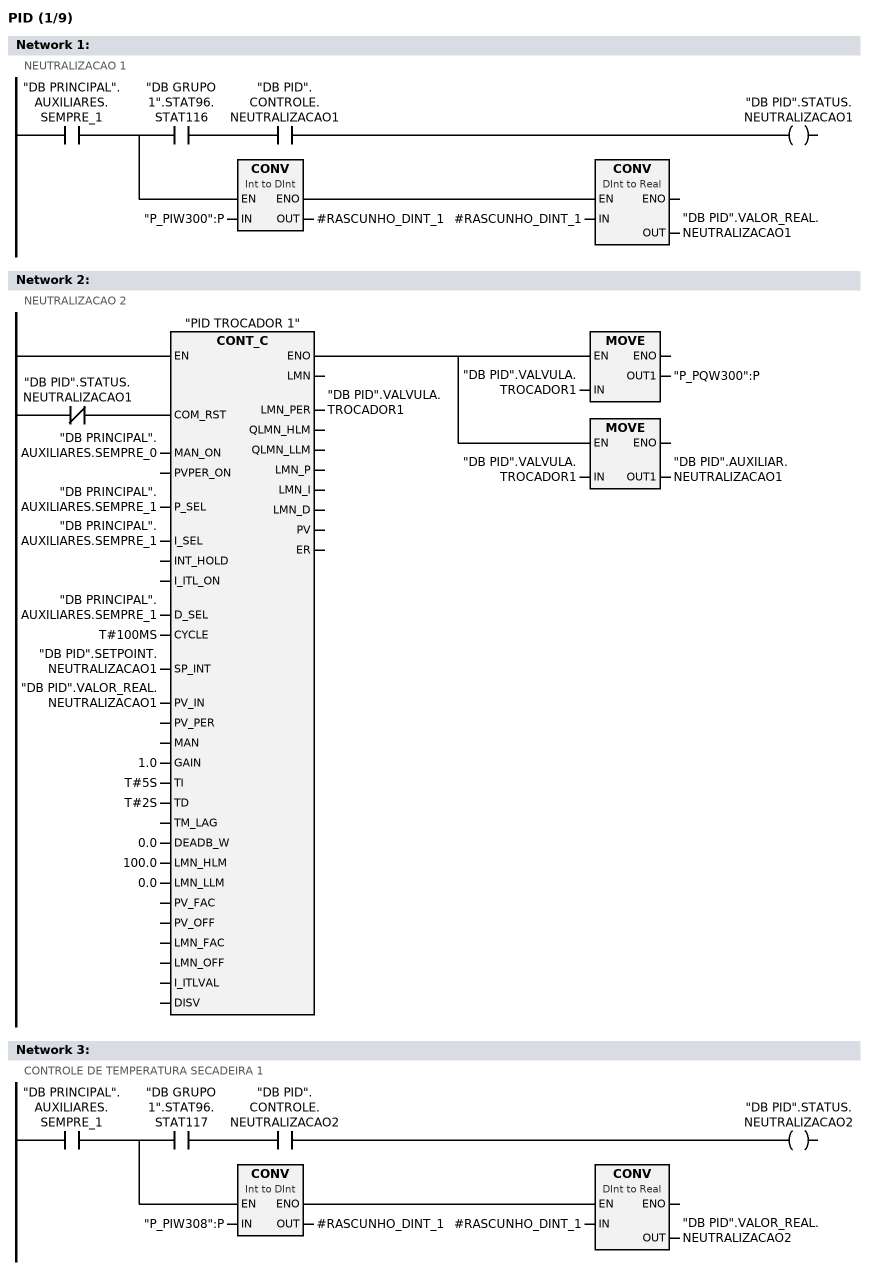
   RUNG wire#powerrail
      Contact( "DB PRINCIPAL".AUXILIARES.SEMPRE_1 )
      wire#w1
      Contact( "DB GRUPO 1".STAT96.STAT116 )
      Contact( "DB PID".CONTROLE.NEUTRALIZACAO1 )
      Coil( "DB PID".STATUS.NEUTRALIZACAO1 )
   END_RUNG
   RUNG wire#w1
      { S7_Templates := "[SrcType := Int, DestType := DInt]"; S7_GenerateENO := "TRUE" } Convert(in := "P_PIW300":P, out => #RASCUNHO_DINT_1)
      { S7_Templates := "[SrcType := DInt, DestType := Real]"; S7_GenerateENO := "TRUE" } Convert(in := #RASCUNHO_DINT_1, out => "DB PID".VALOR_REAL.NEUTRALIZACAO1)
   END_RUNG
   // the same network as SCL:
   // ENO of a box is taken as its EN; it also drops when the box reports an error
   "DB PID".STATUS.NEUTRALIZACAO1 := "DB PRINCIPAL".AUXILIARES.SEMPRE_1 AND "DB GRUPO 1".STAT96.STAT116 AND "DB PID".CONTROLE.NEUTRALIZACAO1;
   IF "DB PRINCIPAL".AUXILIARES.SEMPRE_1 THEN
       #RASCUNHO_DINT_1 := INT_TO_DINT("P_PIW300":P);
       "DB PID".VALOR_REAL.NEUTRALIZACAO1 := DINT_TO_REAL(#RASCUNHO_DINT_1);
   END_IF;
END_REGION

REGION Network 2
   // NEUTRALIZACAO 2
   // ENO of a box is taken as its EN; it also drops when the box reports an error
   "PID TROCADOR 1"(COM_RST := NOT "DB PID".STATUS.NEUTRALIZACAO1,   // CONT_C
                    MAN_ON := "DB PRINCIPAL".AUXILIARES.SEMPRE_0,
                    P_SEL := "DB PRINCIPAL".AUXILIARES.SEMPRE_1,
                    I_SEL := "DB PRINCIPAL".AUXILIARES.SEMPRE_1,
                    D_SEL := "DB PRINCIPAL".AUXILIARES.SEMPRE_1,
                    CYCLE := T#100MS,
                    SP_INT := "DB PID".SETPOINT.NEUTRALIZACAO1,
                    PV_IN := "DB PID".VALOR_REAL.NEUTRALIZACAO1,
                    GAIN := 1.0,
                    TI := T#5S,
                    TD := T#2S,
                    DEADB_W := 0.0,
                    LMN_HLM := 100.0,
                    LMN_LLM := 0.0,
                    LMN_PER => "DB PID".VALVULA.TROCADOR1);
   "P_PQW300":P := "DB PID".VALVULA.TROCADOR1;
   "DB PID".AUXILIAR.NEUTRALIZACAO1 := "DB PID".VALVULA.TROCADOR1;
END_REGION

REGION Network 3
   // CONTROLE DE TEMPERATURA SECADEIRA 1
   RUNG wire#powerrail
      Contact( "DB PRINCIPAL".AUXILIARES.SEMPRE_1 )
      wire#w1
      Contact( "DB GRUPO 1".STAT96.STAT117 )
      Contact( "DB PID".CONTROLE.NEUTRALIZACAO2 )
      Coil( "DB PID".STATUS.NEUTRALIZACAO2 )
   END_RUNG
   RUNG wire#w1
      { S7_Templates := "[SrcType := Int, DestType := DInt]"; S7_GenerateENO := "TRUE" } Convert(in := "P_PIW308":P, out => #RASCUNHO_DINT_1)
      { S7_Templates := "[SrcType := DInt, DestType := Real]"; S7_GenerateENO := "TRUE" } Convert(in := #RASCUNHO_DINT_1, out => "DB PID".VALOR_REAL.NEUTRALIZACAO2)
   END_RUNG
   // the same network as SCL:
   // ENO of a box is taken as its EN; it also drops when the box reports an error
   "DB PID".STATUS.NEUTRALIZACAO2 := "DB PRINCIPAL".AUXILIARES.SEMPRE_1 AND "DB GRUPO 1".STAT96.STAT117 AND "DB PID".CONTROLE.NEUTRALIZACAO2;
   IF "DB PRINCIPAL".AUXILIARES.SEMPRE_1 THEN
       #RASCUNHO_DINT_1 := INT_TO_DINT("P_PIW308":P);
       "DB PID".VALOR_REAL.NEUTRALIZACAO2 := DINT_TO_REAL(#RASCUNHO_DINT_1);
   END_IF;
END_REGION

REGION Network 4
   // CONTROLE DE TEMPERATURA SECADEIRA 2
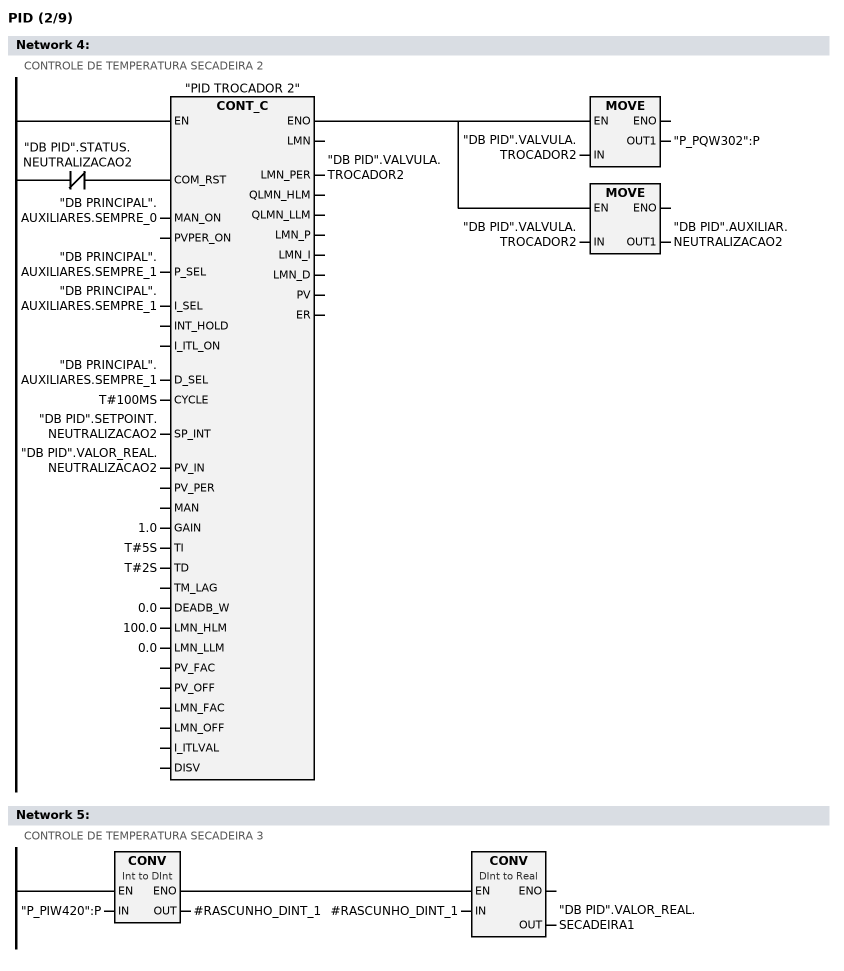
   // ENO of a box is taken as its EN; it also drops when the box reports an error
   "PID TROCADOR 2"(COM_RST := NOT "DB PID".STATUS.NEUTRALIZACAO2,   // CONT_C
                    MAN_ON := "DB PRINCIPAL".AUXILIARES.SEMPRE_0,
                    P_SEL := "DB PRINCIPAL".AUXILIARES.SEMPRE_1,
                    I_SEL := "DB PRINCIPAL".AUXILIARES.SEMPRE_1,
                    D_SEL := "DB PRINCIPAL".AUXILIARES.SEMPRE_1,
                    CYCLE := T#100MS,
                    SP_INT := "DB PID".SETPOINT.NEUTRALIZACAO2,
                    PV_IN := "DB PID".VALOR_REAL.NEUTRALIZACAO2,
                    GAIN := 1.0,
                    TI := T#5S,
                    TD := T#2S,
                    DEADB_W := 0.0,
                    LMN_HLM := 100.0,
                    LMN_LLM := 0.0,
                    LMN_PER => "DB PID".VALVULA.TROCADOR2);
   "P_PQW302":P := "DB PID".VALVULA.TROCADOR2;
   "DB PID".AUXILIAR.NEUTRALIZACAO2 := "DB PID".VALVULA.TROCADOR2;
END_REGION

REGION Network 5
   // CONTROLE DE TEMPERATURA SECADEIRA 3
   RUNG wire#powerrail
      { S7_Templates := "[SrcType := Int, DestType := DInt]"; S7_GenerateENO := "TRUE" } Convert(in := "P_PIW420":P, out => #RASCUNHO_DINT_1)
      { S7_Templates := "[SrcType := DInt, DestType := Real]"; S7_GenerateENO := "TRUE" } Convert(in := #RASCUNHO_DINT_1, out => "DB PID".VALOR_REAL.SECADEIRA1)
   END_RUNG
   // the same network as SCL:
   // ENO of a box is taken as its EN; it also drops when the box reports an error
   #RASCUNHO_DINT_1 := INT_TO_DINT("P_PIW420":P);
   "DB PID".VALOR_REAL.SECADEIRA1 := DINT_TO_REAL(#RASCUNHO_DINT_1);
END_REGION

REGION Network 6
   // CONTROLE DE TEMPERATURA SECADEIRA 4
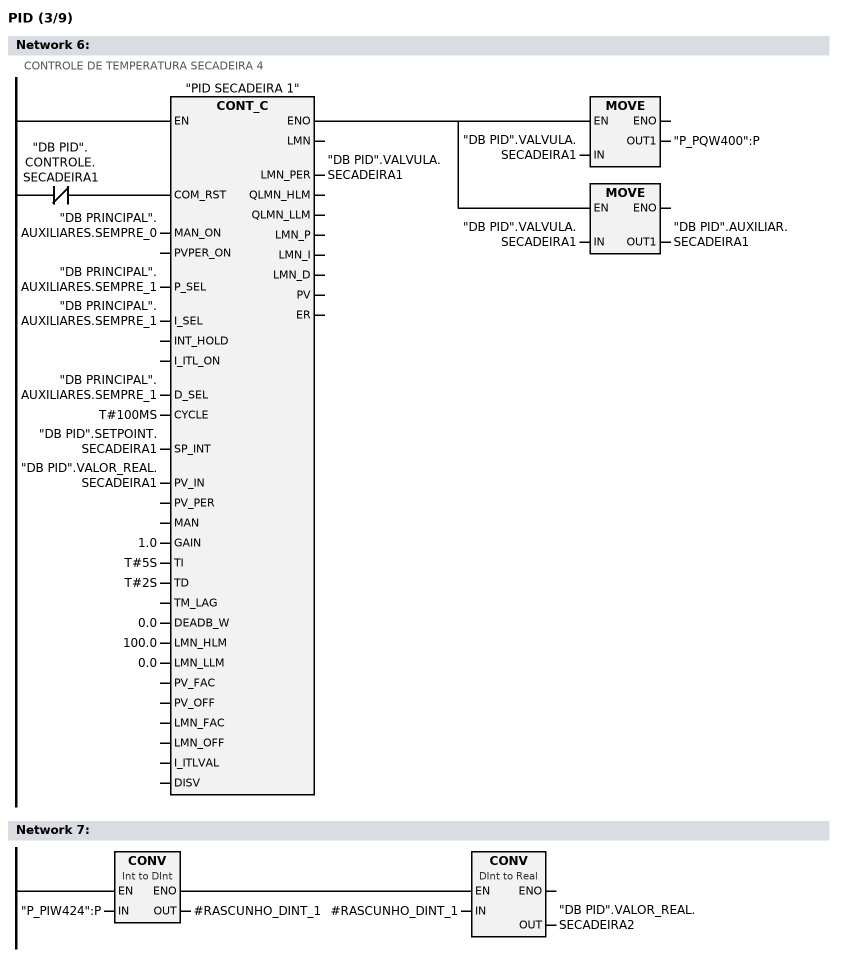
   // ENO of a box is taken as its EN; it also drops when the box reports an error
   "PID SECADEIRA 1"(COM_RST := NOT "DB PID".CONTROLE.SECADEIRA1,   // CONT_C
                     MAN_ON := "DB PRINCIPAL".AUXILIARES.SEMPRE_0,
                     P_SEL := "DB PRINCIPAL".AUXILIARES.SEMPRE_1,
                     I_SEL := "DB PRINCIPAL".AUXILIARES.SEMPRE_1,
                     D_SEL := "DB PRINCIPAL".AUXILIARES.SEMPRE_1,
                     CYCLE := T#100MS,
                     SP_INT := "DB PID".SETPOINT.SECADEIRA1,
                     PV_IN := "DB PID".VALOR_REAL.SECADEIRA1,
                     GAIN := 1.0,
                     TI := T#5S,
                     TD := T#2S,
                     DEADB_W := 0.0,
                     LMN_HLM := 100.0,
                     LMN_LLM := 0.0,
                     LMN_PER => "DB PID".VALVULA.SECADEIRA1);
   "P_PQW400":P := "DB PID".VALVULA.SECADEIRA1;
   "DB PID".AUXILIAR.SECADEIRA1 := "DB PID".VALVULA.SECADEIRA1;
END_REGION

REGION Network 7
   RUNG wire#powerrail
      { S7_Templates := "[SrcType := Int, DestType := DInt]"; S7_GenerateENO := "TRUE" } Convert(in := "P_PIW424":P, out => #RASCUNHO_DINT_1)
      { S7_Templates := "[SrcType := DInt, DestType := Real]"; S7_GenerateENO := "TRUE" } Convert(in := #RASCUNHO_DINT_1, out => "DB PID".VALOR_REAL.SECADEIRA2)
   END_RUNG
   // the same network as SCL:
   // ENO of a box is taken as its EN; it also drops when the box reports an error
   #RASCUNHO_DINT_1 := INT_TO_DINT("P_PIW424":P);
   "DB PID".VALOR_REAL.SECADEIRA2 := DINT_TO_REAL(#RASCUNHO_DINT_1);
END_REGION

REGION Network 8
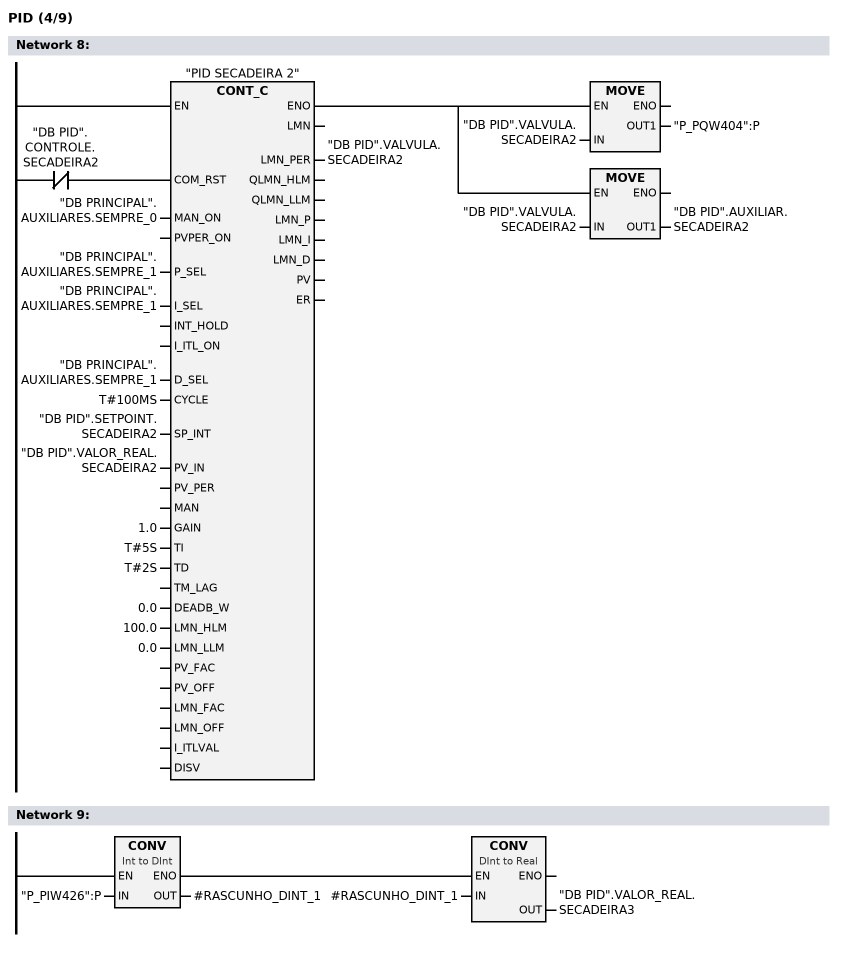
   // ENO of a box is taken as its EN; it also drops when the box reports an error
   "PID SECADEIRA 2"(COM_RST := NOT "DB PID".CONTROLE.SECADEIRA2,   // CONT_C
                     MAN_ON := "DB PRINCIPAL".AUXILIARES.SEMPRE_0,
                     P_SEL := "DB PRINCIPAL".AUXILIARES.SEMPRE_1,
                     I_SEL := "DB PRINCIPAL".AUXILIARES.SEMPRE_1,
                     D_SEL := "DB PRINCIPAL".AUXILIARES.SEMPRE_1,
                     CYCLE := T#100MS,
                     SP_INT := "DB PID".SETPOINT.SECADEIRA2,
                     PV_IN := "DB PID".VALOR_REAL.SECADEIRA2,
                     GAIN := 1.0,
                     TI := T#5S,
                     TD := T#2S,
                     DEADB_W := 0.0,
                     LMN_HLM := 100.0,
                     LMN_LLM := 0.0,
                     LMN_PER => "DB PID".VALVULA.SECADEIRA2);
   "P_PQW404":P := "DB PID".VALVULA.SECADEIRA2;
   "DB PID".AUXILIAR.SECADEIRA2 := "DB PID".VALVULA.SECADEIRA2;
END_REGION

REGION Network 9
   RUNG wire#powerrail
      { S7_Templates := "[SrcType := Int, DestType := DInt]"; S7_GenerateENO := "TRUE" } Convert(in := "P_PIW426":P, out => #RASCUNHO_DINT_1)
      { S7_Templates := "[SrcType := DInt, DestType := Real]"; S7_GenerateENO := "TRUE" } Convert(in := #RASCUNHO_DINT_1, out => "DB PID".VALOR_REAL.SECADEIRA3)
   END_RUNG
   // the same network as SCL:
   // ENO of a box is taken as its EN; it also drops when the box reports an error
   #RASCUNHO_DINT_1 := INT_TO_DINT("P_PIW426":P);
   "DB PID".VALOR_REAL.SECADEIRA3 := DINT_TO_REAL(#RASCUNHO_DINT_1);
END_REGION

REGION Network 10
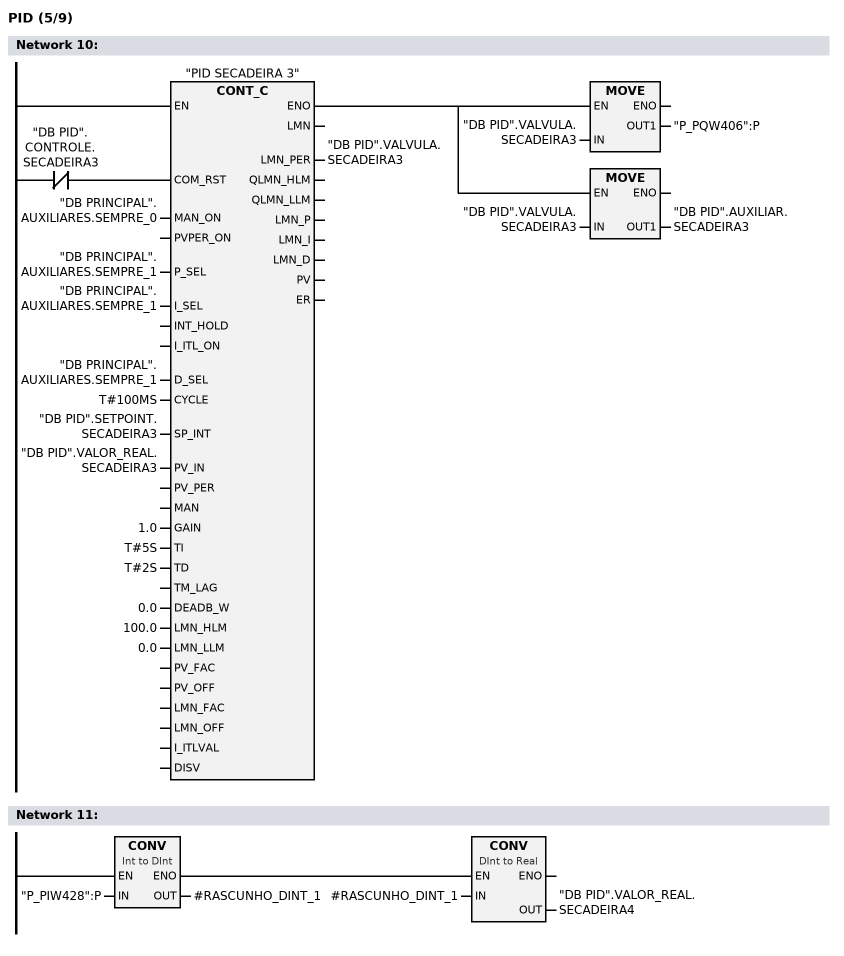
   // ENO of a box is taken as its EN; it also drops when the box reports an error
   "PID SECADEIRA 3"(COM_RST := NOT "DB PID".CONTROLE.SECADEIRA3,   // CONT_C
                     MAN_ON := "DB PRINCIPAL".AUXILIARES.SEMPRE_0,
                     P_SEL := "DB PRINCIPAL".AUXILIARES.SEMPRE_1,
                     I_SEL := "DB PRINCIPAL".AUXILIARES.SEMPRE_1,
                     D_SEL := "DB PRINCIPAL".AUXILIARES.SEMPRE_1,
                     CYCLE := T#100MS,
                     SP_INT := "DB PID".SETPOINT.SECADEIRA3,
                     PV_IN := "DB PID".VALOR_REAL.SECADEIRA3,
                     GAIN := 1.0,
                     TI := T#5S,
                     TD := T#2S,
                     DEADB_W := 0.0,
                     LMN_HLM := 100.0,
                     LMN_LLM := 0.0,
                     LMN_PER => "DB PID".VALVULA.SECADEIRA3);
   "P_PQW406":P := "DB PID".VALVULA.SECADEIRA3;
   "DB PID".AUXILIAR.SECADEIRA3 := "DB PID".VALVULA.SECADEIRA3;
END_REGION

REGION Network 11
   RUNG wire#powerrail
      { S7_Templates := "[SrcType := Int, DestType := DInt]"; S7_GenerateENO := "TRUE" } Convert(in := "P_PIW428":P, out => #RASCUNHO_DINT_1)
      { S7_Templates := "[SrcType := DInt, DestType := Real]"; S7_GenerateENO := "TRUE" } Convert(in := #RASCUNHO_DINT_1, out => "DB PID".VALOR_REAL.SECADEIRA4)
   END_RUNG
   // the same network as SCL:
   // ENO of a box is taken as its EN; it also drops when the box reports an error
   #RASCUNHO_DINT_1 := INT_TO_DINT("P_PIW428":P);
   "DB PID".VALOR_REAL.SECADEIRA4 := DINT_TO_REAL(#RASCUNHO_DINT_1);
END_REGION

REGION Network 12: PID SECADEIRA 4
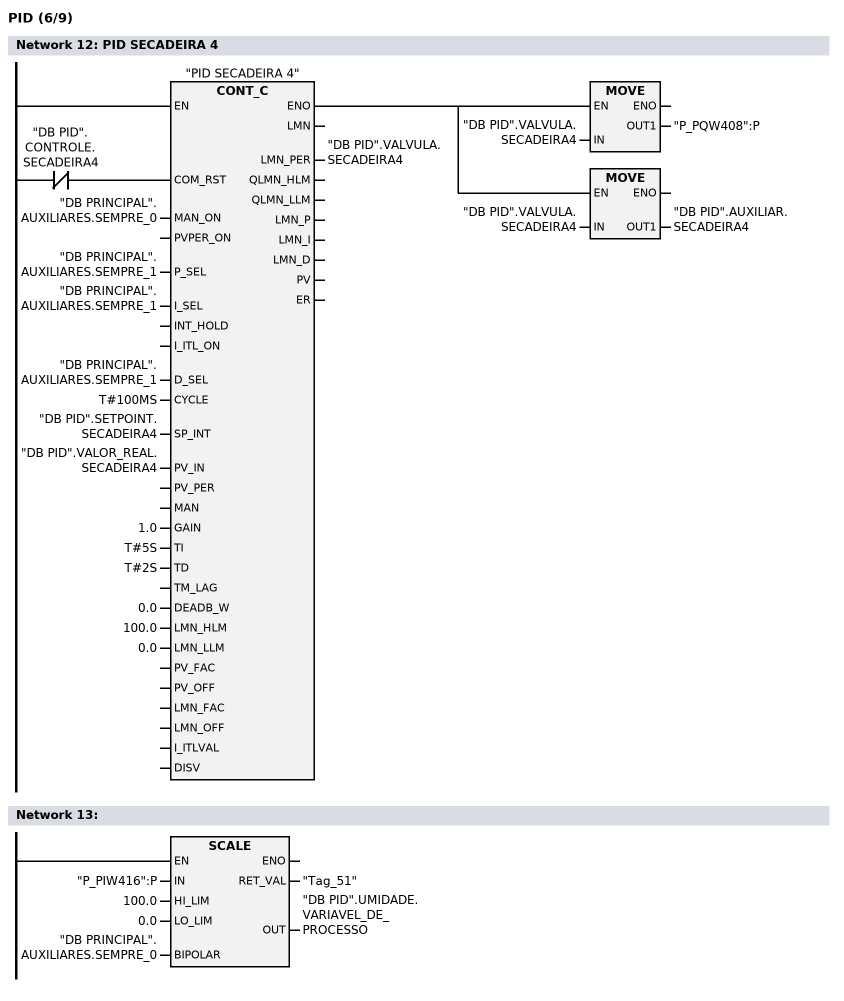
   // ENO of a box is taken as its EN; it also drops when the box reports an error
   "PID SECADEIRA 4"(COM_RST := NOT "DB PID".CONTROLE.SECADEIRA4,   // CONT_C
                     MAN_ON := "DB PRINCIPAL".AUXILIARES.SEMPRE_0,
                     P_SEL := "DB PRINCIPAL".AUXILIARES.SEMPRE_1,
                     I_SEL := "DB PRINCIPAL".AUXILIARES.SEMPRE_1,
                     D_SEL := "DB PRINCIPAL".AUXILIARES.SEMPRE_1,
                     CYCLE := T#100MS,
                     SP_INT := "DB PID".SETPOINT.SECADEIRA4,
                     PV_IN := "DB PID".VALOR_REAL.SECADEIRA4,
                     GAIN := 1.0,
                     TI := T#5S,
                     TD := T#2S,
                     DEADB_W := 0.0,
                     LMN_HLM := 100.0,
                     LMN_LLM := 0.0,
                     LMN_PER => "DB PID".VALVULA.SECADEIRA4);
   "P_PQW408":P := "DB PID".VALVULA.SECADEIRA4;
   "DB PID".AUXILIAR.SECADEIRA4 := "DB PID".VALVULA.SECADEIRA4;
END_REGION

REGION Network 13
   "Tag_51" := SCALE(IN := "P_PIW416":P,
                     HI_LIM := 100.0,
                     LO_LIM := 0.0,
                     BIPOLAR := "DB PRINCIPAL".AUXILIARES.SEMPRE_0,
                     OUT => "DB PID".UMIDADE.VARIAVEL_DE_PROCESSO);
END_REGION

REGION Network 14: PID SECADEIRA 4 - Controle de Umidade
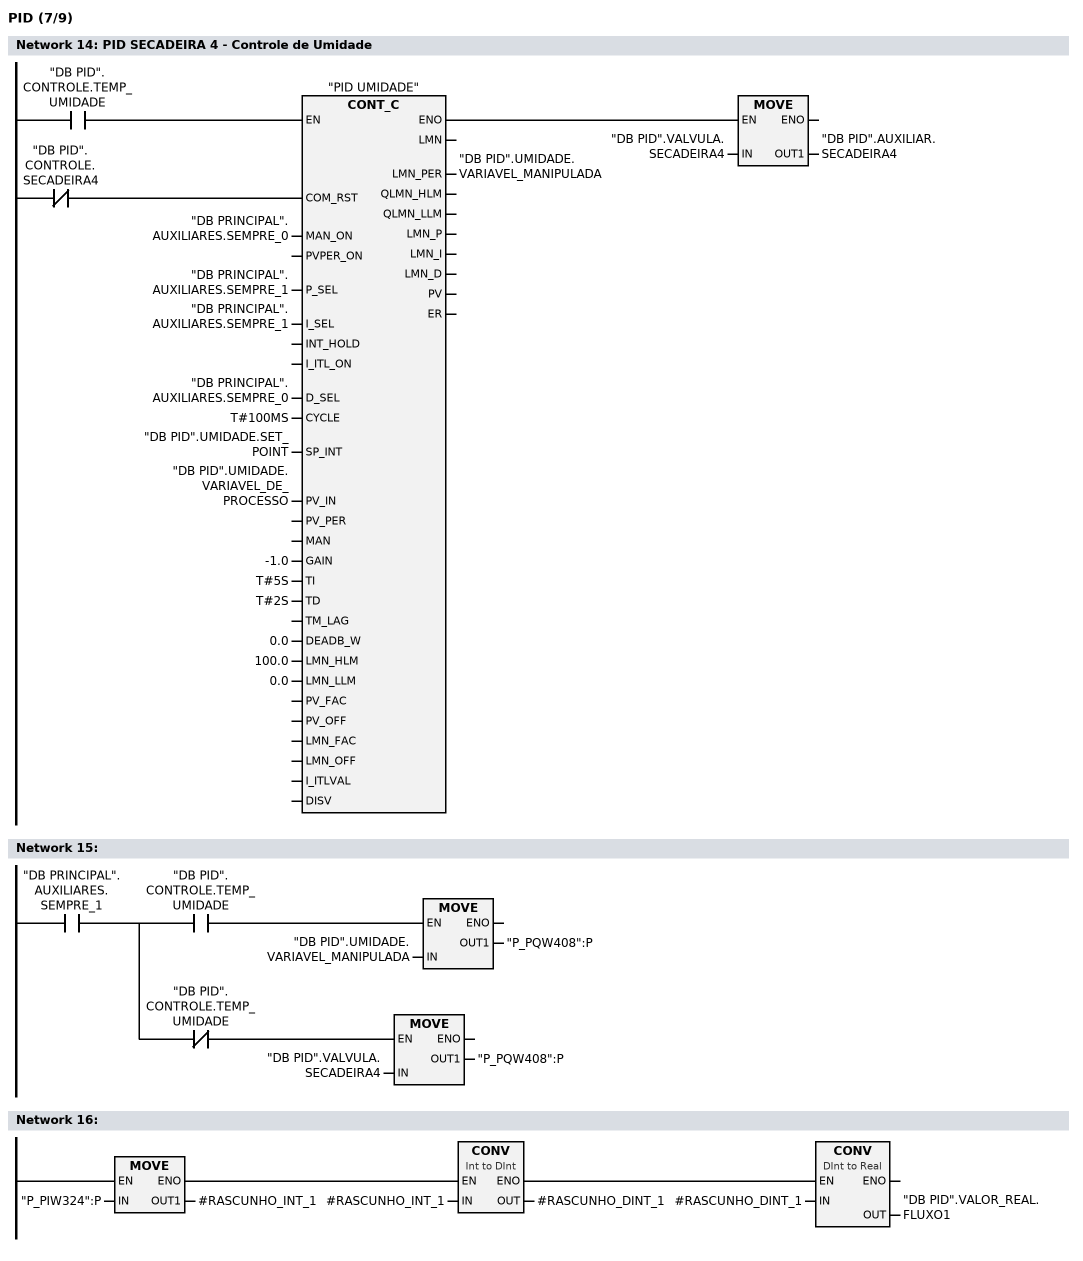
   // ENO of a box is taken as its EN; it also drops when the box reports an error
   #_w1 := "DB PID".CONTROLE.TEMP_UMIDADE;
   IF #_w1 THEN
       "PID UMIDADE"(COM_RST := NOT "DB PID".CONTROLE.SECADEIRA4,   // CONT_C
                     MAN_ON := "DB PRINCIPAL".AUXILIARES.SEMPRE_0,
                     P_SEL := "DB PRINCIPAL".AUXILIARES.SEMPRE_1,
                     I_SEL := "DB PRINCIPAL".AUXILIARES.SEMPRE_1,
                     D_SEL := "DB PRINCIPAL".AUXILIARES.SEMPRE_0,
                     CYCLE := T#100MS,
                     SP_INT := "DB PID".UMIDADE.SET_POINT,
                     PV_IN := "DB PID".UMIDADE.VARIAVEL_DE_PROCESSO,
                     GAIN := -1.0,
                     TI := T#5S,
                     TD := T#2S,
                     DEADB_W := 0.0,
                     LMN_HLM := 100.0,
                     LMN_LLM := 0.0,
                     LMN_PER => "DB PID".UMIDADE.VARIAVEL_MANIPULADA);
       "DB PID".AUXILIAR.SECADEIRA4 := "DB PID".VALVULA.SECADEIRA4;
   END_IF;
END_REGION

REGION Network 15
   RUNG wire#powerrail
      Contact( "DB PRINCIPAL".AUXILIARES.SEMPRE_1 )
      wire#w1
      Contact( "DB PID".CONTROLE.TEMP_UMIDADE )
      { S7_GenerateENO := "TRUE" } Move(in := "DB PID".UMIDADE.VARIAVEL_MANIPULADA, out1 => "P_PQW408":P)
   END_RUNG
   RUNG wire#w1
      I_Contact( "DB PID".CONTROLE.TEMP_UMIDADE )
      { S7_GenerateENO := "TRUE" } Move(in := "DB PID".VALVULA.SECADEIRA4, out1 => "P_PQW408":P)
   END_RUNG
   // the same network as SCL:
   IF "DB PRINCIPAL".AUXILIARES.SEMPRE_1 AND "DB PID".CONTROLE.TEMP_UMIDADE THEN
       "P_PQW408":P := "DB PID".UMIDADE.VARIAVEL_MANIPULADA;
   END_IF;
   IF "DB PRINCIPAL".AUXILIARES.SEMPRE_1 AND NOT "DB PID".CONTROLE.TEMP_UMIDADE THEN
       "P_PQW408":P := "DB PID".VALVULA.SECADEIRA4;
   END_IF;
END_REGION

REGION Network 16
   RUNG wire#powerrail
      { S7_GenerateENO := "TRUE" } Move(in := "P_PIW324":P, out1 => #RASCUNHO_INT_1)
      { S7_Templates := "[SrcType := Int, DestType := DInt]"; S7_GenerateENO := "TRUE" } Convert(in := #RASCUNHO_INT_1, out => #RASCUNHO_DINT_1)
      { S7_Templates := "[SrcType := DInt, DestType := Real]"; S7_GenerateENO := "TRUE" } Convert(in := #RASCUNHO_DINT_1, out => "DB PID".VALOR_REAL.FLUXO1)
   END_RUNG
   // the same network as SCL:
   // ENO of a box is taken as its EN; it also drops when the box reports an error
   #RASCUNHO_INT_1 := "P_PIW324":P;
   #RASCUNHO_DINT_1 := INT_TO_DINT(#RASCUNHO_INT_1);
   "DB PID".VALOR_REAL.FLUXO1 := DINT_TO_REAL(#RASCUNHO_DINT_1);
END_REGION

REGION Network 17
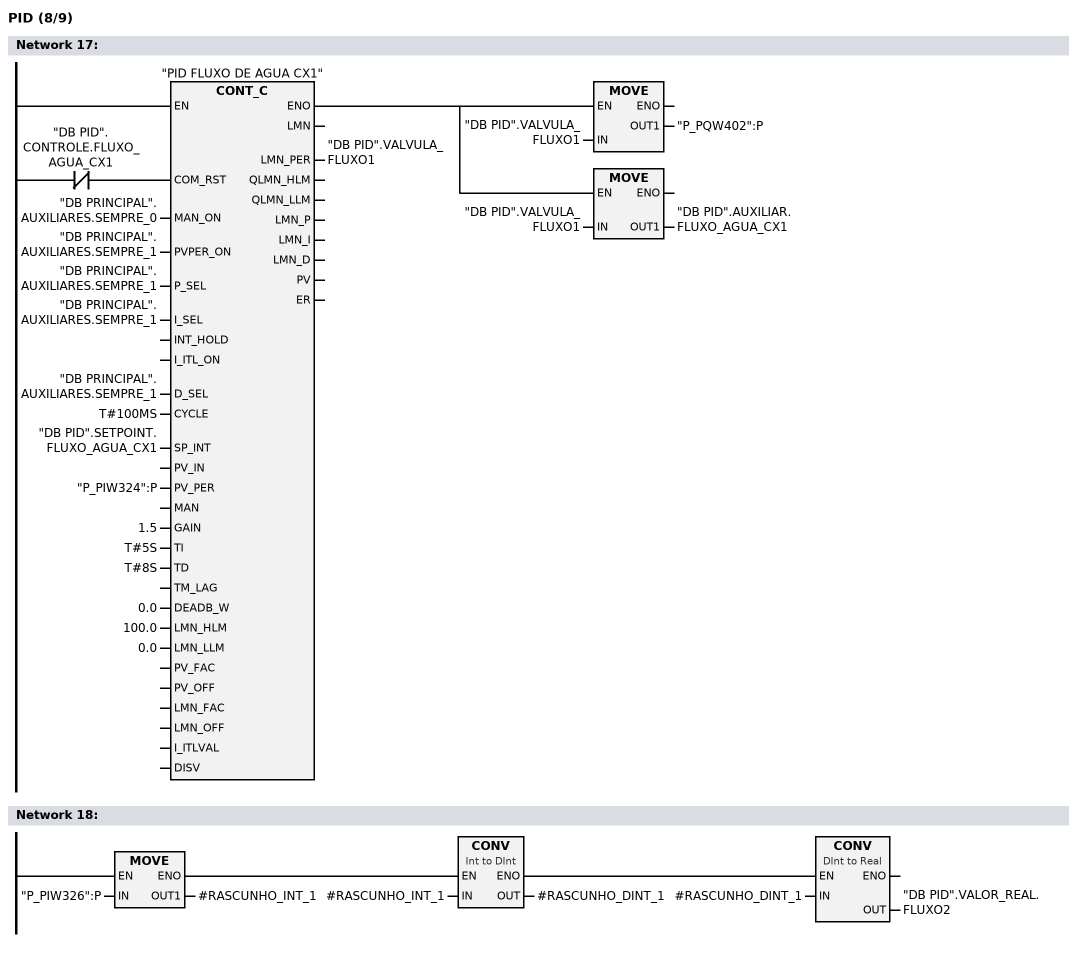
   // ENO of a box is taken as its EN; it also drops when the box reports an error
   "PID FLUXO DE AGUA CX1"(COM_RST := NOT "DB PID".CONTROLE.FLUXO_AGUA_CX1,   // CONT_C
                           MAN_ON := "DB PRINCIPAL".AUXILIARES.SEMPRE_0,
                           PVPER_ON := "DB PRINCIPAL".AUXILIARES.SEMPRE_1,
                           P_SEL := "DB PRINCIPAL".AUXILIARES.SEMPRE_1,
                           I_SEL := "DB PRINCIPAL".AUXILIARES.SEMPRE_1,
                           D_SEL := "DB PRINCIPAL".AUXILIARES.SEMPRE_1,
                           CYCLE := T#100MS,
                           SP_INT := "DB PID".SETPOINT.FLUXO_AGUA_CX1,
                           PV_PER := "P_PIW324":P,
                           GAIN := 1.5,
                           TI := T#5S,
                           TD := T#8S,
                           DEADB_W := 0.0,
                           LMN_HLM := 100.0,
                           LMN_LLM := 0.0,
                           LMN_PER => "DB PID".VALVULA_FLUXO1);
   "P_PQW402":P := "DB PID".VALVULA_FLUXO1;
   "DB PID".AUXILIAR.FLUXO_AGUA_CX1 := "DB PID".VALVULA_FLUXO1;
END_REGION

REGION Network 18
   RUNG wire#powerrail
      { S7_GenerateENO := "TRUE" } Move(in := "P_PIW326":P, out1 => #RASCUNHO_INT_1)
      { S7_Templates := "[SrcType := Int, DestType := DInt]"; S7_GenerateENO := "TRUE" } Convert(in := #RASCUNHO_INT_1, out => #RASCUNHO_DINT_1)
      { S7_Templates := "[SrcType := DInt, DestType := Real]"; S7_GenerateENO := "TRUE" } Convert(in := #RASCUNHO_DINT_1, out => "DB PID".VALOR_REAL.FLUXO2)
   END_RUNG
   // the same network as SCL:
   // ENO of a box is taken as its EN; it also drops when the box reports an error
   #RASCUNHO_INT_1 := "P_PIW326":P;
   #RASCUNHO_DINT_1 := INT_TO_DINT(#RASCUNHO_INT_1);
   "DB PID".VALOR_REAL.FLUXO2 := DINT_TO_REAL(#RASCUNHO_DINT_1);
END_REGION

REGION Network 19
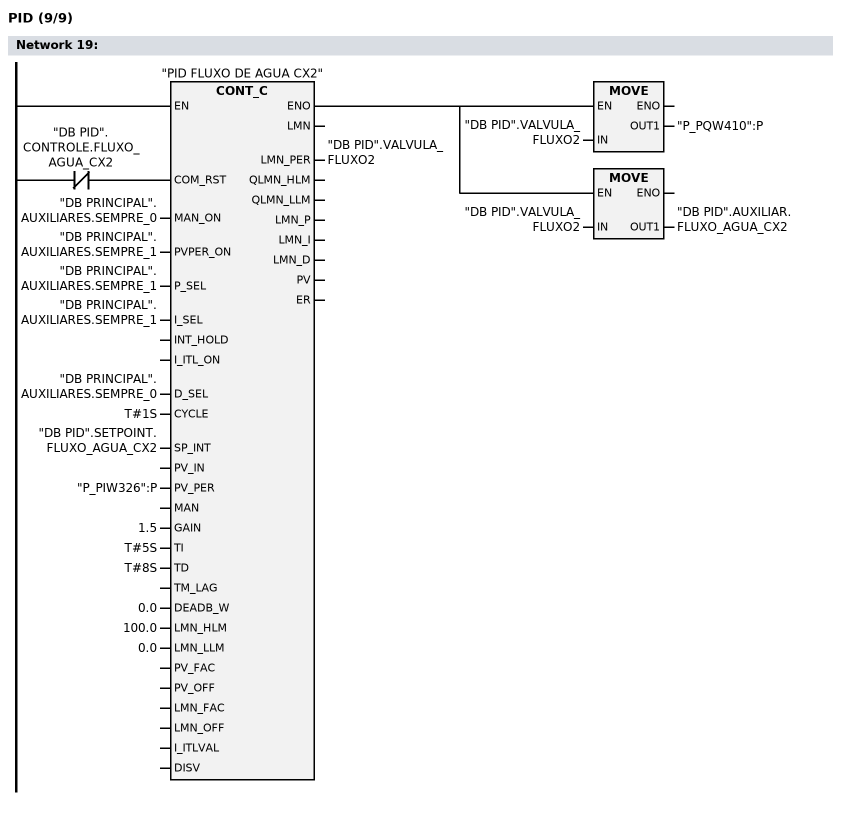
   // ENO of a box is taken as its EN; it also drops when the box reports an error
   "PID FLUXO DE AGUA CX2"(COM_RST := NOT "DB PID".CONTROLE.FLUXO_AGUA_CX2,   // CONT_C
                           MAN_ON := "DB PRINCIPAL".AUXILIARES.SEMPRE_0,
                           PVPER_ON := "DB PRINCIPAL".AUXILIARES.SEMPRE_1,
                           P_SEL := "DB PRINCIPAL".AUXILIARES.SEMPRE_1,
                           I_SEL := "DB PRINCIPAL".AUXILIARES.SEMPRE_1,
                           D_SEL := "DB PRINCIPAL".AUXILIARES.SEMPRE_0,
                           CYCLE := T#1S,
                           SP_INT := "DB PID".SETPOINT.FLUXO_AGUA_CX2,
                           PV_PER := "P_PIW326":P,
                           GAIN := 1.5,
                           TI := T#5S,
                           TD := T#8S,
                           DEADB_W := 0.0,
                           LMN_HLM := 100.0,
                           LMN_LLM := 0.0,
                           LMN_PER => "DB PID".VALVULA_FLUXO2);
   "P_PQW410":P := "DB PID".VALVULA_FLUXO2;
   "DB PID".AUXILIAR.FLUXO_AGUA_CX2 := "DB PID".VALVULA_FLUXO2;
END_REGION
END_FUNCTION

FUNCTION "MT_PUXADOR" : Void   // FC10, LAD
TITLE = MÓDULO DE CONTROLE DO PUXADOR DE ENTRADA
{ S7_Optimized_Access := 'FALSE' }
AUTHOR : THALLES
FAMILY : TRAÇÃO
NAME : LINHA
VERSION : 0.1
// DATA BLOCK DE CONTROLE // DB10
// Automation Pack Automação Indl. e Com. Ltda.
// Cliente: Texima S/A Ind. de Máquinas
// Cliente Final: Cia. Fiação e Tecidos Santo Antonio.
// Máquina: Sanforizadeira Linha 1 - O.S.: 24.626
   VAR_TEMP
      aux_r : Real;
   END_VAR
   VAR_TEMP   // added for the SCL form of the ladder/FBD networks
      _w1 : Bool;
      _w2 : Bool;
      _w3 : Bool;
   END_VAR
BEGIN

REGION Network 1: ALARMES
   // RESET DOS ALARMES
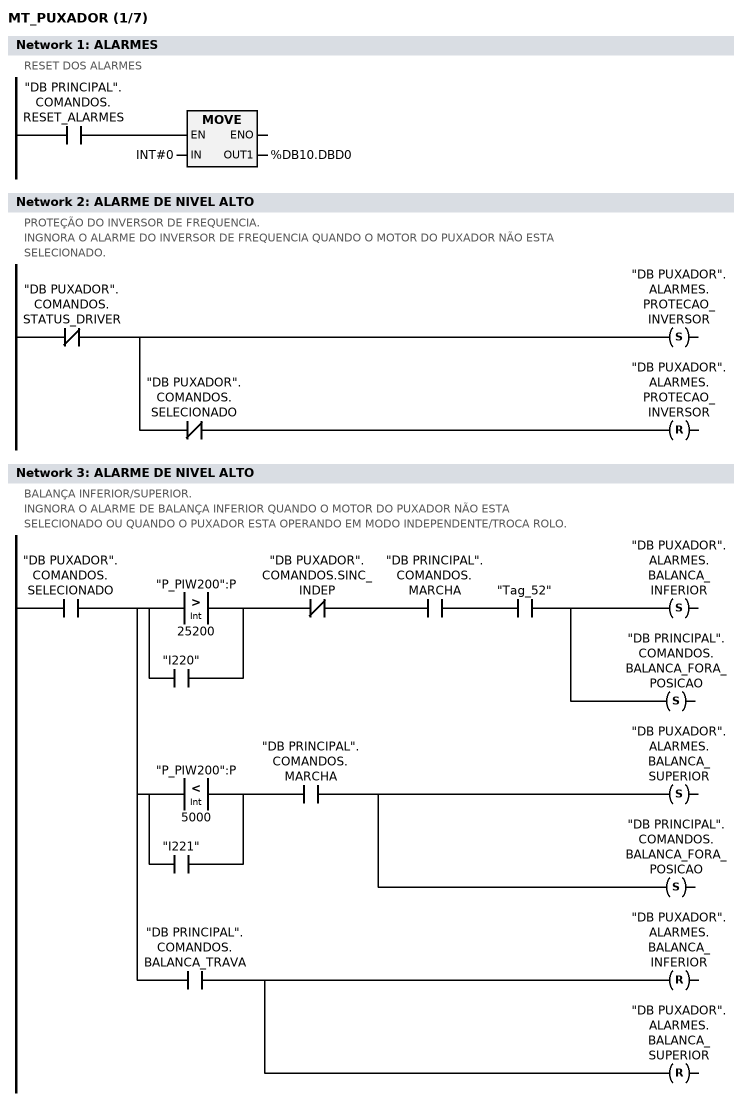
   RUNG wire#powerrail
      Contact( "DB PRINCIPAL".COMANDOS.RESET_ALARMES )
      { S7_GenerateENO := "TRUE" } Move(in := INT#0, out1 => %DB10.DBD0)
   END_RUNG
   // the same network as SCL:
   IF "DB PRINCIPAL".COMANDOS.RESET_ALARMES THEN %DB10.DBD0 := INT#0; END_IF;
END_REGION

REGION Network 2: ALARME DE NIVEL ALTO
   // PROTEÇÃO DO INVERSOR DE FREQUENCIA.
   // INGNORA O ALARME DO INVERSOR DE FREQUENCIA QUANDO O MOTOR DO PUXADOR NÃO ESTA 
   // SELECIONADO.
   RUNG wire#powerrail
      I_Contact( "DB PUXADOR".COMANDOS.STATUS_DRIVER )
      wire#w1
      S_Coil( "DB PUXADOR".ALARMES.PROTECAO_INVERSOR )
   END_RUNG
   RUNG wire#w1
      I_Contact( "DB PUXADOR".COMANDOS.SELECIONADO )
      R_Coil( "DB PUXADOR".ALARMES.PROTECAO_INVERSOR )
   END_RUNG
   // the same network as SCL:
   #_w1 := NOT "DB PUXADOR".COMANDOS.STATUS_DRIVER;
   IF #_w1 THEN "DB PUXADOR".ALARMES.PROTECAO_INVERSOR := TRUE; END_IF;
   IF #_w1 AND NOT "DB PUXADOR".COMANDOS.SELECIONADO THEN
       "DB PUXADOR".ALARMES.PROTECAO_INVERSOR := FALSE;
   END_IF;
END_REGION

REGION Network 3: ALARME DE NIVEL ALTO
   // BALANÇA INFERIOR/SUPERIOR.
   // INGNORA O ALARME DE BALANÇA INFERIOR QUANDO O MOTOR DO PUXADOR NÃO ESTA 
   // SELECIONADO OU QUANDO O PUXADOR ESTA OPERANDO EM MODO INDEPENDENTE/TROCA ROLO.
   RUNG wire#powerrail
      Contact( "DB PUXADOR".COMANDOS.SELECIONADO )
      wire#w1
      { S7_Templates := "SrcType := Int" } GT_Contact(in1 := "P_PIW200":P, in2 := 25200)
      wire#w2
      I_Contact( "DB PUXADOR".COMANDOS.SINC_INDEP )
      Contact( "DB PRINCIPAL".COMANDOS.MARCHA )
      Contact( "Tag_52" )
      wire#w3
      S_Coil( "DB PUXADOR".ALARMES.BALANCA_INFERIOR )
   END_RUNG
   RUNG wire#w1
      Contact( "I220" )
   END_RUNG wire#w2
   RUNG wire#w3
      S_Coil( "DB PRINCIPAL".COMANDOS.BALANCA_FORA_POSICAO )
   END_RUNG
   RUNG wire#w1
      { S7_Templates := "SrcType := Int" } LT_Contact(in1 := "P_PIW200":P, in2 := 5000)
      wire#w4
      Contact( "DB PRINCIPAL".COMANDOS.MARCHA )
      wire#w5
      S_Coil( "DB PUXADOR".ALARMES.BALANCA_SUPERIOR )
   END_RUNG
   RUNG wire#w1
      Contact( "I221" )
   END_RUNG wire#w4
   RUNG wire#w5
      S_Coil( "DB PRINCIPAL".COMANDOS.BALANCA_FORA_POSICAO )
   END_RUNG
   RUNG wire#w1
      Contact( "DB PRINCIPAL".COMANDOS.BALANCA_TRAVA )
      wire#w6
      R_Coil( "DB PUXADOR".ALARMES.BALANCA_INFERIOR )
   END_RUNG
   RUNG wire#w6
      R_Coil( "DB PUXADOR".ALARMES.BALANCA_SUPERIOR )
   END_RUNG
   // the same network as SCL:
   IF "DB PUXADOR".COMANDOS.SELECIONADO AND (("P_PIW200":P > 25200) OR "I220") AND NOT "DB PUXADOR".COMANDOS.SINC_INDEP AND "DB PRINCIPAL".COMANDOS.MARCHA AND "Tag_52" THEN
       "DB PUXADOR".ALARMES.BALANCA_INFERIOR := TRUE;
       "DB PRINCIPAL".COMANDOS.BALANCA_FORA_POSICAO := TRUE;
   END_IF;
   IF "DB PUXADOR".COMANDOS.SELECIONADO AND (("P_PIW200":P < 5000) OR "I221") AND "DB PRINCIPAL".COMANDOS.MARCHA THEN
       "DB PUXADOR".ALARMES.BALANCA_SUPERIOR := TRUE;
       "DB PRINCIPAL".COMANDOS.BALANCA_FORA_POSICAO := TRUE;
   END_IF;
   IF "DB PUXADOR".COMANDOS.SELECIONADO AND "DB PRINCIPAL".COMANDOS.BALANCA_TRAVA THEN
       "DB PUXADOR".ALARMES.BALANCA_INFERIOR := FALSE;
       "DB PUXADOR".ALARMES.BALANCA_SUPERIOR := FALSE;
   END_IF;
END_REGION

REGION Network 4: ALARMES
   // ATIVAÇÃO DO BIT DE ALARME DE NIVEL ALTO.
   // ATIVAÇÃO DO BIT DE ALARME DE NIVEL BAIXO.
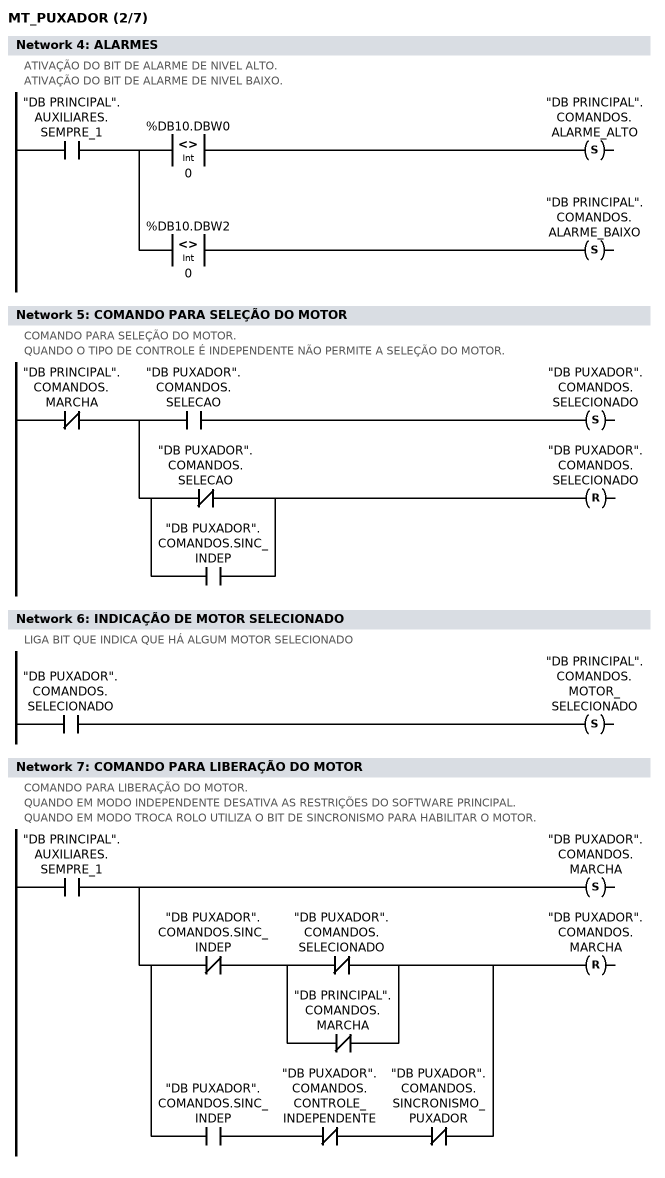
   RUNG wire#powerrail
      Contact( "DB PRINCIPAL".AUXILIARES.SEMPRE_1 )
      wire#w1
      { S7_Templates := "SrcType := Int" } NE_Contact(in1 := %DB10.DBW0, in2 := 0)
      S_Coil( "DB PRINCIPAL".COMANDOS.ALARME_ALTO )
   END_RUNG
   RUNG wire#w1
      { S7_Templates := "SrcType := Int" } NE_Contact(in1 := %DB10.DBW2, in2 := 0)
      S_Coil( "DB PRINCIPAL".COMANDOS.ALARME_BAIXO )
   END_RUNG
   // the same network as SCL:
   IF "DB PRINCIPAL".AUXILIARES.SEMPRE_1 AND (%DB10.DBW0 <> 0) THEN
       "DB PRINCIPAL".COMANDOS.ALARME_ALTO := TRUE;
   END_IF;
   IF "DB PRINCIPAL".AUXILIARES.SEMPRE_1 AND (%DB10.DBW2 <> 0) THEN
       "DB PRINCIPAL".COMANDOS.ALARME_BAIXO := TRUE;
   END_IF;
END_REGION

REGION Network 5: COMANDO PARA SELEÇÃO DO MOTOR
   // COMANDO PARA SELEÇÃO DO MOTOR. 
   // QUANDO O TIPO DE CONTROLE É INDEPENDENTE NÃO PERMITE A SELEÇÃO DO MOTOR.
   RUNG wire#powerrail
      I_Contact( "DB PRINCIPAL".COMANDOS.MARCHA )
      wire#w1
      Contact( "DB PUXADOR".COMANDOS.SELECAO )
      S_Coil( "DB PUXADOR".COMANDOS.SELECIONADO )
   END_RUNG
   RUNG wire#w1
      I_Contact( "DB PUXADOR".COMANDOS.SELECAO )
      wire#w2
      R_Coil( "DB PUXADOR".COMANDOS.SELECIONADO )
   END_RUNG
   RUNG wire#w1
      Contact( "DB PUXADOR".COMANDOS.SINC_INDEP )
   END_RUNG wire#w2
   // the same network as SCL:
   #_w1 := NOT "DB PRINCIPAL".COMANDOS.MARCHA;
   IF #_w1 AND "DB PUXADOR".COMANDOS.SELECAO THEN "DB PUXADOR".COMANDOS.SELECIONADO := TRUE; END_IF;
   IF #_w1 AND (NOT "DB PUXADOR".COMANDOS.SELECAO OR "DB PUXADOR".COMANDOS.SINC_INDEP) THEN
       "DB PUXADOR".COMANDOS.SELECIONADO := FALSE;
   END_IF;
END_REGION

REGION Network 6: INDICAÇÃO DE MOTOR SELECIONADO
   // LIGA BIT QUE INDICA QUE HÁ ALGUM MOTOR SELECIONADO
   RUNG wire#powerrail
      Contact( "DB PUXADOR".COMANDOS.SELECIONADO )
      S_Coil( "DB PRINCIPAL".COMANDOS.MOTOR_SELECIONADO )
   END_RUNG
   // the same network as SCL:
   IF "DB PUXADOR".COMANDOS.SELECIONADO THEN "DB PRINCIPAL".COMANDOS.MOTOR_SELECIONADO := TRUE; END_IF;
END_REGION

REGION Network 7: COMANDO PARA LIBERAÇÃO DO MOTOR
   // COMANDO PARA LIBERAÇÃO DO MOTOR.
   // QUANDO EM MODO INDEPENDENTE DESATIVA AS RESTRIÇÕES DO SOFTWARE PRINCIPAL.
   // QUANDO EM MODO TROCA ROLO UTILIZA O BIT DE SINCRONISMO PARA HABILITAR O MOTOR.
   RUNG wire#powerrail
      Contact( "DB PRINCIPAL".AUXILIARES.SEMPRE_1 )
      wire#w1
      S_Coil( "DB PUXADOR".COMANDOS.MARCHA )
   END_RUNG
   RUNG wire#w1
      I_Contact( "DB PUXADOR".COMANDOS.SINC_INDEP )
      wire#w2
      I_Contact( "DB PUXADOR".COMANDOS.SELECIONADO )
      wire#w3
      R_Coil( "DB PUXADOR".COMANDOS.MARCHA )
   END_RUNG
   RUNG wire#w2
      I_Contact( "DB PRINCIPAL".COMANDOS.MARCHA )
   END_RUNG wire#w3
   RUNG wire#w1
      Contact( "DB PUXADOR".COMANDOS.SINC_INDEP )
      I_Contact( "DB PUXADOR".COMANDOS.CONTROLE_INDEPENDENTE )
      I_Contact( "DB PUXADOR".COMANDOS.SINCRONISMO_PUXADOR )
   END_RUNG wire#w3
   // the same network as SCL:
   IF "DB PRINCIPAL".AUXILIARES.SEMPRE_1 THEN "DB PUXADOR".COMANDOS.MARCHA := TRUE; END_IF;
   IF "DB PRINCIPAL".AUXILIARES.SEMPRE_1 AND ((NOT "DB PUXADOR".COMANDOS.SINC_INDEP AND (NOT "DB PUXADOR".COMANDOS.SELECIONADO OR NOT "DB PRINCIPAL".COMANDOS.MARCHA)) OR ("DB PUXADOR".COMANDOS.SINC_INDEP AND NOT "DB PUXADOR".COMANDOS.CONTROLE_INDEPENDENTE AND NOT "DB PUXADOR".COMANDOS.SINCRONISMO_PUXADOR)) THEN
       "DB PUXADOR".COMANDOS.MARCHA := FALSE;
   END_IF;
END_REGION

REGION Network 8: JOG DO MOTOR
   // JOG DO MOTOR
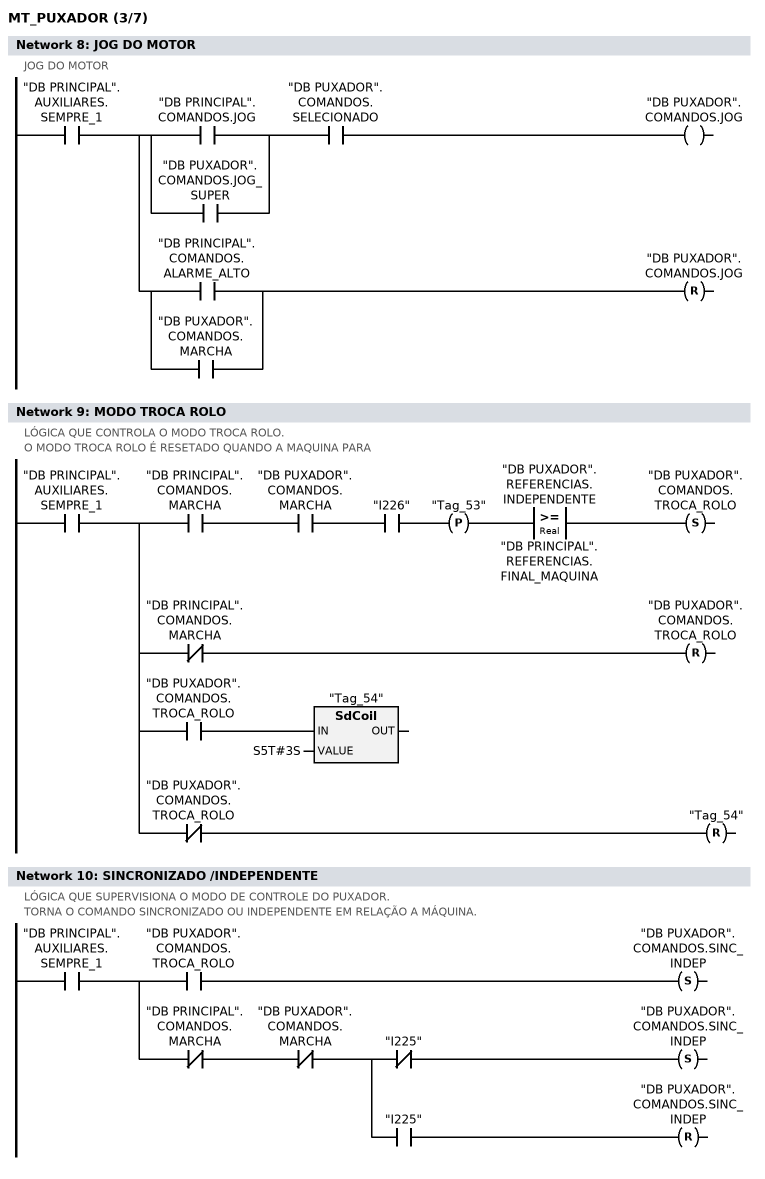
   RUNG wire#powerrail
      Contact( "DB PRINCIPAL".AUXILIARES.SEMPRE_1 )
      wire#w1
      Contact( "DB PRINCIPAL".COMANDOS.JOG )
      wire#w2
      Contact( "DB PUXADOR".COMANDOS.SELECIONADO )
      Coil( "DB PUXADOR".COMANDOS.JOG )
   END_RUNG
   RUNG wire#w1
      Contact( "DB PUXADOR".COMANDOS.JOG_SUPER )
   END_RUNG wire#w2
   RUNG wire#w1
      Contact( "DB PRINCIPAL".COMANDOS.ALARME_ALTO )
      wire#w3
      R_Coil( "DB PUXADOR".COMANDOS.JOG )
   END_RUNG
   RUNG wire#w1
      Contact( "DB PUXADOR".COMANDOS.MARCHA )
   END_RUNG wire#w3
   // the same network as SCL:
   "DB PUXADOR".COMANDOS.JOG := "DB PRINCIPAL".AUXILIARES.SEMPRE_1 AND ("DB PRINCIPAL".COMANDOS.JOG OR "DB PUXADOR".COMANDOS.JOG_SUPER) AND "DB PUXADOR".COMANDOS.SELECIONADO;
   IF "DB PRINCIPAL".AUXILIARES.SEMPRE_1 AND ("DB PRINCIPAL".COMANDOS.ALARME_ALTO OR "DB PUXADOR".COMANDOS.MARCHA) THEN
       "DB PUXADOR".COMANDOS.JOG := FALSE;
   END_IF;
END_REGION

REGION Network 9: MODO TROCA ROLO
   // LÓGICA QUE CONTROLA O MODO TROCA ROLO.
   // O MODO TROCA ROLO É RESETADO QUANDO A MAQUINA PARA
   // no SCL statement known for SdCoil: written as a call
   #_w1 := "DB PRINCIPAL".AUXILIARES.SEMPRE_1 AND "DB PRINCIPAL".COMANDOS.MARCHA AND "DB PUXADOR".COMANDOS.MARCHA AND "I226";
   #_w2 := #_w1 AND NOT "Tag_53";   // rising edge
   "Tag_53" := #_w1;
   IF #_w2 AND ("DB PUXADOR".REFERENCIAS.INDEPENDENTE >= "DB PRINCIPAL".REFERENCIAS.FINAL_MAQUINA) THEN
       "DB PUXADOR".COMANDOS.TROCA_ROLO := TRUE;
   END_IF;
   IF "DB PRINCIPAL".AUXILIARES.SEMPRE_1 AND NOT "DB PRINCIPAL".COMANDOS.MARCHA THEN
       "DB PUXADOR".COMANDOS.TROCA_ROLO := FALSE;
   END_IF;
   #_w3 := "DB PRINCIPAL".AUXILIARES.SEMPRE_1;
   SdCoil(value := S5T#3S,
          operand := "Tag_54",
          in := "DB PRINCIPAL".AUXILIARES.SEMPRE_1 AND "DB PUXADOR".COMANDOS.TROCA_ROLO);
   IF #_w3 AND NOT "DB PUXADOR".COMANDOS.TROCA_ROLO THEN "Tag_54" := FALSE; END_IF;
END_REGION

REGION Network 10: SINCRONIZADO /INDEPENDENTE
   // LÓGICA QUE SUPERVISIONA O MODO DE CONTROLE DO PUXADOR.
   // TORNA O COMANDO SINCRONIZADO OU INDEPENDENTE EM RELAÇÃO A MÁQUINA.
   RUNG wire#powerrail
      Contact( "DB PRINCIPAL".AUXILIARES.SEMPRE_1 )
      wire#w1
      Contact( "DB PUXADOR".COMANDOS.TROCA_ROLO )
      S_Coil( "DB PUXADOR".COMANDOS.SINC_INDEP )
   END_RUNG
   RUNG wire#w1
      I_Contact( "DB PRINCIPAL".COMANDOS.MARCHA )
      I_Contact( "DB PUXADOR".COMANDOS.MARCHA )
      wire#w2
      I_Contact( "I225" )
      S_Coil( "DB PUXADOR".COMANDOS.SINC_INDEP )
   END_RUNG
   RUNG wire#w2
      Contact( "I225" )
      R_Coil( "DB PUXADOR".COMANDOS.SINC_INDEP )
   END_RUNG
   // the same network as SCL:
   IF "DB PRINCIPAL".AUXILIARES.SEMPRE_1 AND "DB PUXADOR".COMANDOS.TROCA_ROLO THEN
       "DB PUXADOR".COMANDOS.SINC_INDEP := TRUE;
   END_IF;
   #_w1 := "DB PRINCIPAL".AUXILIARES.SEMPRE_1 AND NOT "DB PRINCIPAL".COMANDOS.MARCHA AND NOT "DB PUXADOR".COMANDOS.MARCHA;
   IF #_w1 AND NOT "I225" THEN "DB PUXADOR".COMANDOS.SINC_INDEP := TRUE; END_IF;
   IF #_w1 AND "I225" THEN "DB PUXADOR".COMANDOS.SINC_INDEP := FALSE; END_IF;
END_REGION

REGION Network 11: COMANDO INDEPENDENTE
   // LÓGICA DE LIGA / DESLIGA O PUXADOR EM MODO INDEPENDENTE.
   // NO MODO TROCA ROLO O PRÓPRIO BIT DO TROCA ROLO FAZ A FUNÇÃO DE BOTÃO LIGA.
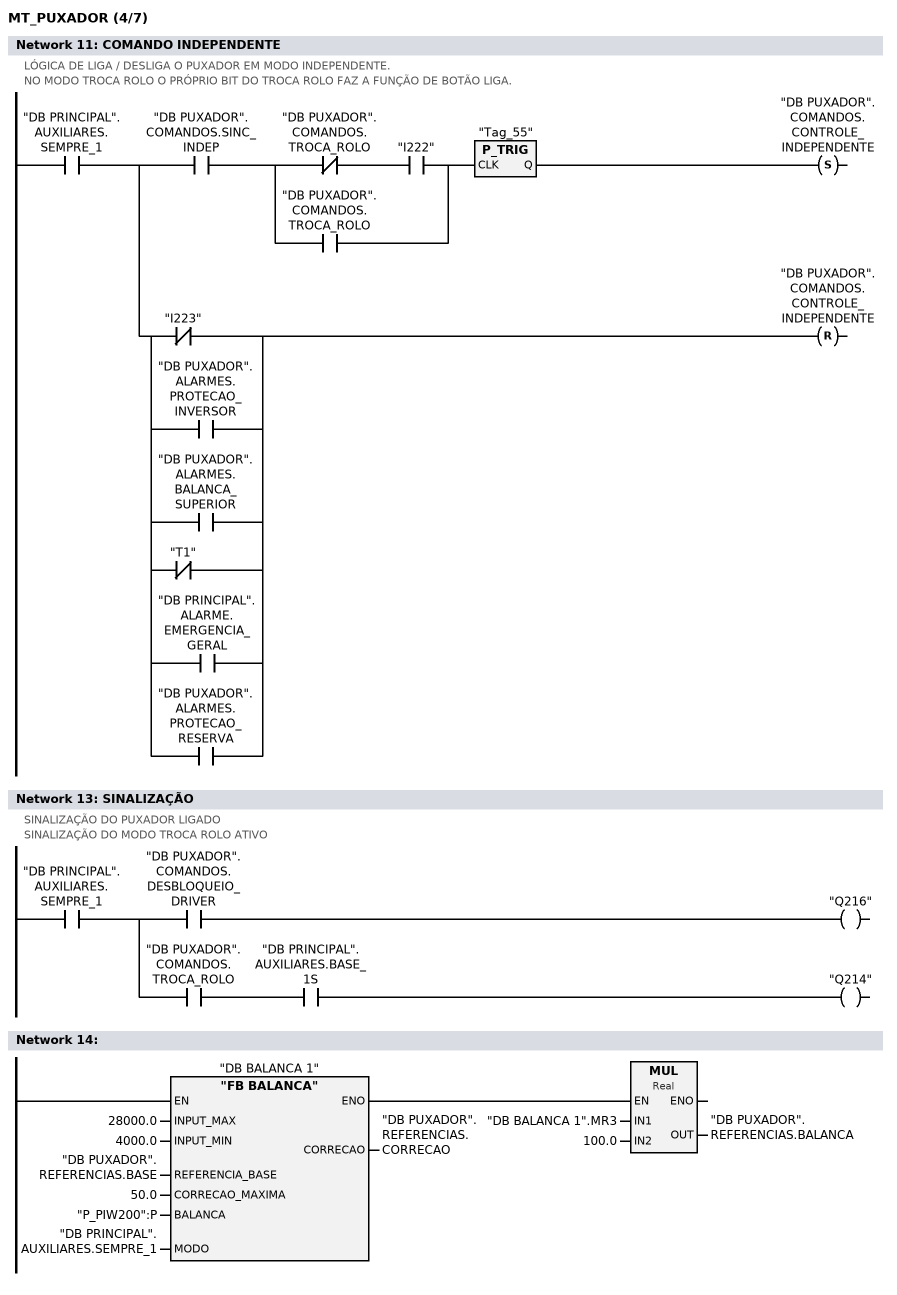
   RUNG wire#powerrail
      Contact( "DB PRINCIPAL".AUXILIARES.SEMPRE_1 )
      wire#w1
      Contact( "DB PUXADOR".COMANDOS.SINC_INDEP )
      wire#w2
      I_Contact( "DB PUXADOR".COMANDOS.TROCA_ROLO )
      Contact( "I222" )
      wire#w3
      P_Trig( "Tag_55" )
      S_Coil( "DB PUXADOR".COMANDOS.CONTROLE_INDEPENDENTE )
   END_RUNG
   RUNG wire#w2
      Contact( "DB PUXADOR".COMANDOS.TROCA_ROLO )
   END_RUNG wire#w3
   RUNG wire#w1
      I_Contact( "I223" )
      wire#w4
      R_Coil( "DB PUXADOR".COMANDOS.CONTROLE_INDEPENDENTE )
   END_RUNG
   RUNG wire#w1
      Contact( "DB PUXADOR".ALARMES.PROTECAO_INVERSOR )
   END_RUNG wire#w4
   RUNG wire#w1
      Contact( "DB PUXADOR".ALARMES.BALANCA_SUPERIOR )
   END_RUNG wire#w4
   RUNG wire#w1
      I_Contact( "T1" )
   END_RUNG wire#w4
   RUNG wire#w1
      Contact( "DB PRINCIPAL".ALARME.EMERGENCIA_GERAL )
   END_RUNG wire#w4
   RUNG wire#w1
      Contact( "DB PUXADOR".ALARMES.PROTECAO_RESERVA )
   END_RUNG wire#w4
   // the same network as SCL:
   #_w1 := "DB PRINCIPAL".AUXILIARES.SEMPRE_1 AND "DB PUXADOR".COMANDOS.SINC_INDEP AND ((NOT "DB PUXADOR".COMANDOS.TROCA_ROLO AND "I222") OR "DB PUXADOR".COMANDOS.TROCA_ROLO);
   #_w2 := #_w1 AND NOT "Tag_55";   // rising edge
   "Tag_55" := #_w1;
   IF #_w2 THEN "DB PUXADOR".COMANDOS.CONTROLE_INDEPENDENTE := TRUE; END_IF;
   IF "DB PRINCIPAL".AUXILIARES.SEMPRE_1 AND (NOT "I223" OR "DB PUXADOR".ALARMES.PROTECAO_INVERSOR OR "DB PUXADOR".ALARMES.BALANCA_SUPERIOR OR NOT "T1" OR "DB PRINCIPAL".ALARME.EMERGENCIA_GERAL OR "DB PUXADOR".ALARMES.PROTECAO_RESERVA) THEN
       "DB PUXADOR".COMANDOS.CONTROLE_INDEPENDENTE := FALSE;
   END_IF;
END_REGION

REGION Network 12 (STL): SINCRONISMO PUXADOR
   // SINCRONIZA O PUXADOR COM A MÁQUINA APOS A OPERAÇÃO TROCA ROLO.
   // HABILITA A REFERÊNCIA DO PROGRAMA PRINCIPAL MAIS TAXA DA BALANÇA.
   // APOS A BALANÇA SAIR DA ZONA DE ALARME (95%) RESETA O BIT DE SINCRONISMO, O BIT 
   // DE TROCA ROLO E O BIT DE TIPO DE CONTROLE.
         A     "DB PRINCIPAL".AUXILIARES.SEMPRE_1;
         =     %L25.0;
         A     %L25.0;
         A     "Tag_54";
         A(;
         A     "DB PUXADOR".COMANDOS.CONTROLE_INDEPENDENTE;
         A     "I222";
         O(;
         L     "DB PUXADOR".REFERENCIAS.BALANCA;
         L     70.0;
         <R;
         );
         );
         R     "DB PUXADOR".COMANDOS.SINCRONISMO_PUXADOR;
         R     "DB PUXADOR".COMANDOS.TROCA_ROLO;
         R     "DB PUXADOR".COMANDOS.SINC_INDEP;
         R     "DB PUXADOR".COMANDOS.CONTROLE_INDEPENDENTE;
         S     "DB PUXADOR".COMANDOS.SINCRONISMO_PUXADOR;
         A     %L25.0;
         AN    "DB PRINCIPAL".COMANDOS.MARCHA;
         R     "DB PUXADOR".COMANDOS.SINCRONISMO_PUXADOR;
         A     %L25.0;
         AN    "DB PUXADOR".COMANDOS.SINCRONISMO_PUXADOR;
         L     S5T#3S;
         SD    "Tag_52";
         A     %L25.0;
         A     "DB PUXADOR".COMANDOS.SINCRONISMO_PUXADOR;
         R     "Tag_52";
END_REGION

REGION Network 13: SINALIZAÇÃO
   // SINALIZAÇÃO DO PUXADOR LIGADO
   // SINALIZAÇÃO DO MODO TROCA ROLO ATIVO
   RUNG wire#powerrail
      Contact( "DB PRINCIPAL".AUXILIARES.SEMPRE_1 )
      wire#w1
      Contact( "DB PUXADOR".COMANDOS.DESBLOQUEIO_DRIVER )
      Coil( "Q216" )
   END_RUNG
   RUNG wire#w1
      Contact( "DB PUXADOR".COMANDOS.TROCA_ROLO )
      Contact( "DB PRINCIPAL".AUXILIARES.BASE_1S )
      Coil( "Q214" )
   END_RUNG
   // the same network as SCL:
   "Q216" := "DB PRINCIPAL".AUXILIARES.SEMPRE_1 AND "DB PUXADOR".COMANDOS.DESBLOQUEIO_DRIVER;
   "Q214" := "DB PRINCIPAL".AUXILIARES.SEMPRE_1 AND "DB PUXADOR".COMANDOS.TROCA_ROLO AND "DB PRINCIPAL".AUXILIARES.BASE_1S;
END_REGION

REGION Network 14
   RUNG wire#powerrail
      "DB BALANCA 1"(INPUT_MAX := 28000.0, INPUT_MIN := 4000.0, REFERENCIA_BASE := "DB PUXADOR".REFERENCIAS.BASE, CORRECAO_MAXIMA := 50.0, BALANCA := "P_PIW200":P, MODO := "DB PRINCIPAL".AUXILIARES.SEMPRE_1, CORRECAO => "DB PUXADOR".REFERENCIAS.CORRECAO)
      { S7_Templates := "SrcType := Real"; S7_GenerateENO := "TRUE" } Mul(in1 := "DB BALANCA 1".MR3, in2 := 100.0, out => "DB PUXADOR".REFERENCIAS.BALANCA)
   END_RUNG
   // the same network as SCL:
   "DB BALANCA 1"(INPUT_MAX := 28000.0,   // "FB BALANCA"
                  INPUT_MIN := 4000.0,
                  REFERENCIA_BASE := "DB PUXADOR".REFERENCIAS.BASE,
                  CORRECAO_MAXIMA := 50.0,
                  BALANCA := "P_PIW200":P,
                  MODO := "DB PRINCIPAL".AUXILIARES.SEMPRE_1,
                  CORRECAO => "DB PUXADOR".REFERENCIAS.CORRECAO,
                  ENO => #_w1);
   IF #_w1 THEN "DB PUXADOR".REFERENCIAS.BALANCA := "DB BALANCA 1".MR3 * 100.0; END_IF;
END_REGION

REGION Network 15: REFERÊNCIA BASE E MÁXIMA PARA CALCULO DE VELOCIDADE DO MOTOR
   // REFERÊNCIA BASE PARA CALCULO DE VELOCIDADE DO MOTOR
   // CALCULO DA REFERÊNCIA MÁXIMA DO MOTOR DO PUXADOR
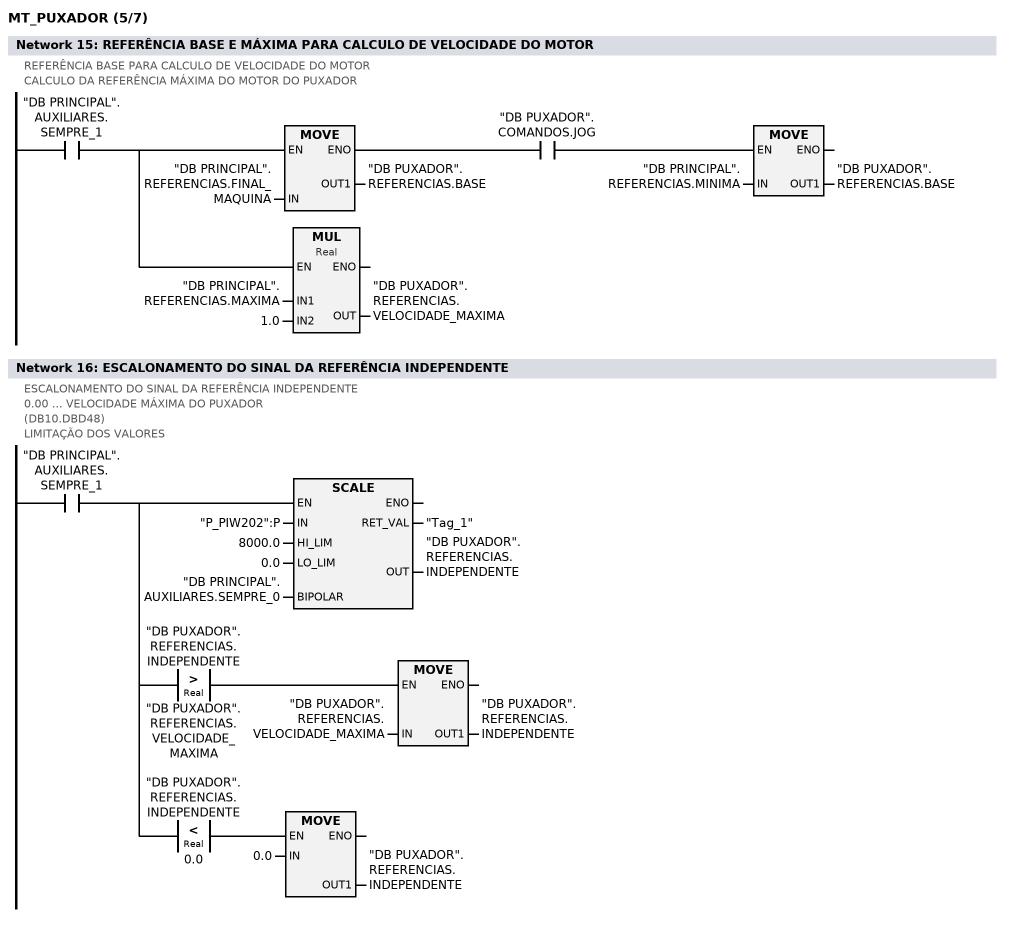
   RUNG wire#powerrail
      Contact( "DB PRINCIPAL".AUXILIARES.SEMPRE_1 )
      wire#w1
      { S7_GenerateENO := "TRUE" } Move(in := "DB PRINCIPAL".REFERENCIAS.FINAL_MAQUINA, out1 => "DB PUXADOR".REFERENCIAS.BASE)
      Contact( "DB PUXADOR".COMANDOS.JOG )
      { S7_GenerateENO := "TRUE" } Move(in := "DB PRINCIPAL".REFERENCIAS.MINIMA, out1 => "DB PUXADOR".REFERENCIAS.BASE)
   END_RUNG
   RUNG wire#w1
      { S7_Templates := "SrcType := Real"; S7_GenerateENO := "TRUE" } Mul(in1 := "DB PRINCIPAL".REFERENCIAS.MAXIMA, in2 := 1.0, out => "DB PUXADOR".REFERENCIAS.VELOCIDADE_MAXIMA)
   END_RUNG
   // the same network as SCL:
   // ENO of a box is taken as its EN; it also drops when the box reports an error
   IF "DB PRINCIPAL".AUXILIARES.SEMPRE_1 THEN
       "DB PUXADOR".REFERENCIAS.BASE := "DB PRINCIPAL".REFERENCIAS.FINAL_MAQUINA;
   END_IF;
   IF "DB PRINCIPAL".AUXILIARES.SEMPRE_1 AND "DB PUXADOR".COMANDOS.JOG THEN
       "DB PUXADOR".REFERENCIAS.BASE := "DB PRINCIPAL".REFERENCIAS.MINIMA;
   END_IF;
   IF "DB PRINCIPAL".AUXILIARES.SEMPRE_1 THEN
       "DB PUXADOR".REFERENCIAS.VELOCIDADE_MAXIMA := "DB PRINCIPAL".REFERENCIAS.MAXIMA * 1.0;
   END_IF;
END_REGION

REGION Network 16: ESCALONAMENTO DO SINAL DA REFERÊNCIA INDEPENDENTE
   // ESCALONAMENTO DO SINAL DA REFERÊNCIA INDEPENDENTE
   // 0.00 ... VELOCIDADE MÁXIMA DO PUXADOR 
   // (DB10.DBD48)
   // LIMITAÇÃO DOS VALORES
   #_w1 := "DB PRINCIPAL".AUXILIARES.SEMPRE_1;
   IF #_w1 THEN
       "Tag_1" := SCALE(IN := "P_PIW202":P,
                        HI_LIM := 8000.0,
                        LO_LIM := 0.0,
                        BIPOLAR := "DB PRINCIPAL".AUXILIARES.SEMPRE_0,
                        OUT => "DB PUXADOR".REFERENCIAS.INDEPENDENTE);
   END_IF;
   IF #_w1 AND ("DB PUXADOR".REFERENCIAS.INDEPENDENTE > "DB PUXADOR".REFERENCIAS.VELOCIDADE_MAXIMA) THEN
       "DB PUXADOR".REFERENCIAS.INDEPENDENTE := "DB PUXADOR".REFERENCIAS.VELOCIDADE_MAXIMA;
   END_IF;
   IF #_w1 AND ("DB PUXADOR".REFERENCIAS.INDEPENDENTE < 0.0) THEN
       "DB PUXADOR".REFERENCIAS.INDEPENDENTE := 0.0;
   END_IF;
END_REGION

REGION Network 17: CALCULO DE REFERÊNCIA PARA O MOTOR
   // REFERÊNCIA MAIS ATÉ 20% DA VELOCIDADE BASE MAXIMA DE CORREÇÃO DA BALANÇA X 
   // REFERÊNCIA INDEPENDENTE
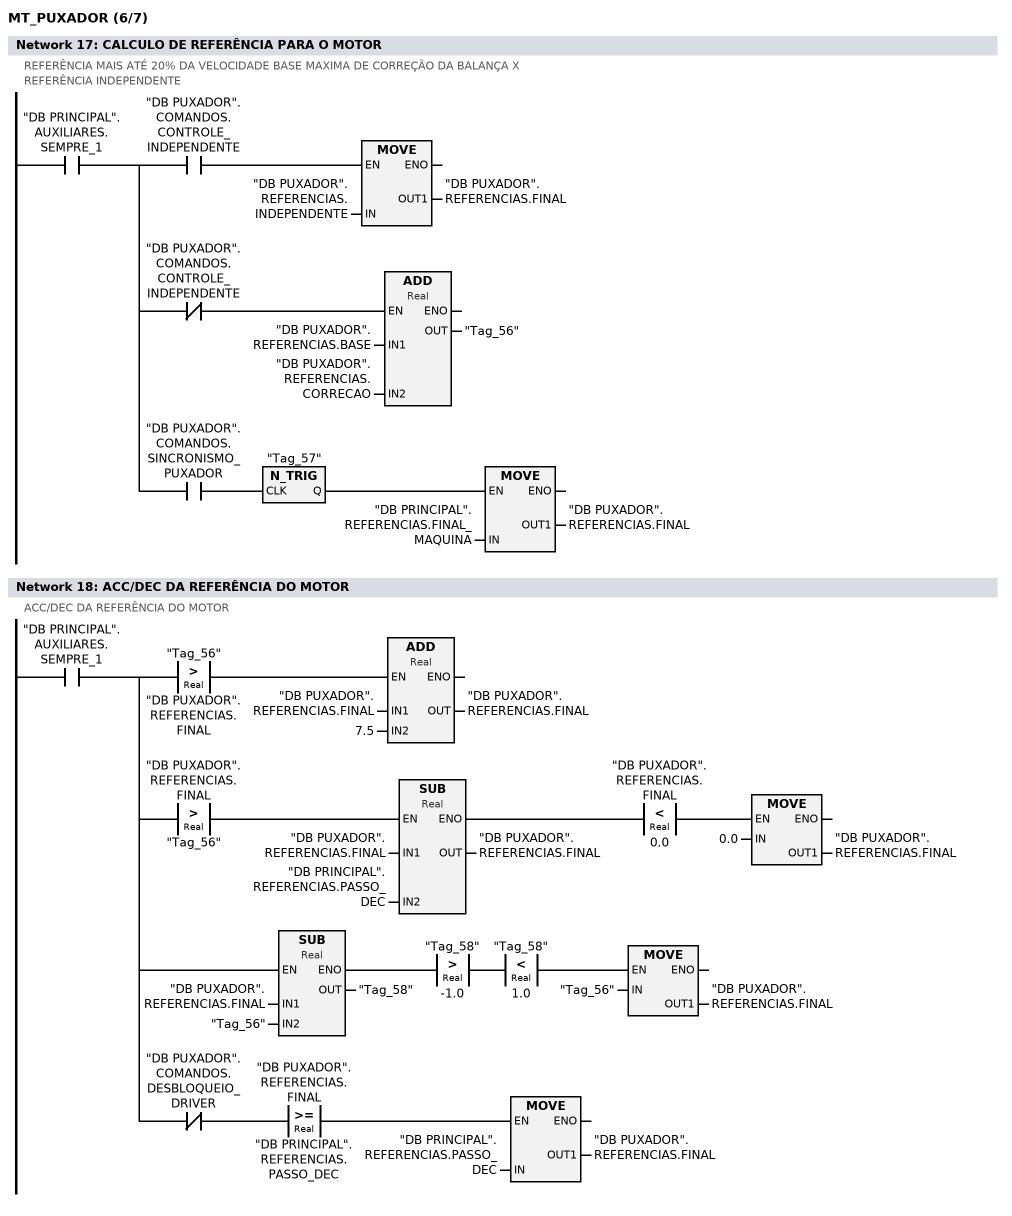
   RUNG wire#powerrail
      Contact( "DB PRINCIPAL".AUXILIARES.SEMPRE_1 )
      wire#w1
      Contact( "DB PUXADOR".COMANDOS.CONTROLE_INDEPENDENTE )
      { S7_GenerateENO := "TRUE" } Move(in := "DB PUXADOR".REFERENCIAS.INDEPENDENTE, out1 => "DB PUXADOR".REFERENCIAS.FINAL)
   END_RUNG
   RUNG wire#w1
      I_Contact( "DB PUXADOR".COMANDOS.CONTROLE_INDEPENDENTE )
      { S7_Templates := "SrcType := Real"; S7_GenerateENO := "TRUE" } Add(in1 := "DB PUXADOR".REFERENCIAS.BASE, in2 := "DB PUXADOR".REFERENCIAS.CORRECAO, out => "Tag_56")
   END_RUNG
   RUNG wire#w1
      Contact( "DB PUXADOR".COMANDOS.SINCRONISMO_PUXADOR )
      N_Trig( "Tag_57" )
      { S7_GenerateENO := "TRUE" } Move(in := "DB PRINCIPAL".REFERENCIAS.FINAL_MAQUINA, out1 => "DB PUXADOR".REFERENCIAS.FINAL)
   END_RUNG
   // the same network as SCL:
   IF "DB PRINCIPAL".AUXILIARES.SEMPRE_1 AND "DB PUXADOR".COMANDOS.CONTROLE_INDEPENDENTE THEN
       "DB PUXADOR".REFERENCIAS.FINAL := "DB PUXADOR".REFERENCIAS.INDEPENDENTE;
   END_IF;
   IF "DB PRINCIPAL".AUXILIARES.SEMPRE_1 AND NOT "DB PUXADOR".COMANDOS.CONTROLE_INDEPENDENTE THEN
       "Tag_56" := "DB PUXADOR".REFERENCIAS.BASE + "DB PUXADOR".REFERENCIAS.CORRECAO;
   END_IF;
   #_w1 := "DB PRINCIPAL".AUXILIARES.SEMPRE_1 AND "DB PUXADOR".COMANDOS.SINCRONISMO_PUXADOR;
   #_w2 := NOT #_w1 AND "Tag_57";   // falling edge
   "Tag_57" := #_w1;
   IF #_w2 THEN "DB PUXADOR".REFERENCIAS.FINAL := "DB PRINCIPAL".REFERENCIAS.FINAL_MAQUINA; END_IF;
END_REGION

REGION Network 18: ACC/DEC DA REFERÊNCIA DO MOTOR
   // ACC/DEC DA REFERÊNCIA DO MOTOR
   RUNG wire#powerrail
      Contact( "DB PRINCIPAL".AUXILIARES.SEMPRE_1 )
      wire#w1
      { S7_Templates := "SrcType := Real" } GT_Contact(in1 := "Tag_56", in2 := "DB PUXADOR".REFERENCIAS.FINAL)
      { S7_Templates := "SrcType := Real"; S7_GenerateENO := "TRUE" } Add(in1 := "DB PUXADOR".REFERENCIAS.FINAL, in2 := 7.5, out => "DB PUXADOR".REFERENCIAS.FINAL)
   END_RUNG
   RUNG wire#w1
      { S7_Templates := "SrcType := Real" } GT_Contact(in1 := "DB PUXADOR".REFERENCIAS.FINAL, in2 := "Tag_56")
      { S7_Templates := "SrcType := Real"; S7_GenerateENO := "TRUE" } Sub(in1 := "DB PUXADOR".REFERENCIAS.FINAL, in2 := "DB PRINCIPAL".REFERENCIAS.PASSO_DEC, out => "DB PUXADOR".REFERENCIAS.FINAL)
      { S7_Templates := "SrcType := Real" } LT_Contact(in1 := "DB PUXADOR".REFERENCIAS.FINAL, in2 := 0.0)
      { S7_GenerateENO := "TRUE" } Move(in := 0.0, out1 => "DB PUXADOR".REFERENCIAS.FINAL)
   END_RUNG
   RUNG wire#w1
      { S7_Templates := "SrcType := Real"; S7_GenerateENO := "TRUE" } Sub(in1 := "DB PUXADOR".REFERENCIAS.FINAL, in2 := "Tag_56", out => "Tag_58")
      { S7_Templates := "SrcType := Real" } GT_Contact(in1 := "Tag_58", in2 := -1.0)
      { S7_Templates := "SrcType := Real" } LT_Contact(in1 := "Tag_58", in2 := 1.0)
      { S7_GenerateENO := "TRUE" } Move(in := "Tag_56", out1 => "DB PUXADOR".REFERENCIAS.FINAL)
   END_RUNG
   RUNG wire#w1
      I_Contact( "DB PUXADOR".COMANDOS.DESBLOQUEIO_DRIVER )
      { S7_Templates := "SrcType := Real" } GE_Contact(in1 := "DB PUXADOR".REFERENCIAS.FINAL, in2 := "DB PRINCIPAL".REFERENCIAS.PASSO_DEC)
      { S7_GenerateENO := "TRUE" } Move(in := "DB PRINCIPAL".REFERENCIAS.PASSO_DEC, out1 => "DB PUXADOR".REFERENCIAS.FINAL)
   END_RUNG
   // the same network as SCL:
   // ENO of a box is taken as its EN; it also drops when the box reports an error
   IF "DB PRINCIPAL".AUXILIARES.SEMPRE_1 AND ("Tag_56" > "DB PUXADOR".REFERENCIAS.FINAL) THEN
       "DB PUXADOR".REFERENCIAS.FINAL := "DB PUXADOR".REFERENCIAS.FINAL + 7.5;
   END_IF;
   #_w1 := "DB PRINCIPAL".AUXILIARES.SEMPRE_1 AND ("DB PUXADOR".REFERENCIAS.FINAL > "Tag_56");
   IF #_w1 THEN
       "DB PUXADOR".REFERENCIAS.FINAL := "DB PUXADOR".REFERENCIAS.FINAL - "DB PRINCIPAL".REFERENCIAS.PASSO_DEC;
   END_IF;
   IF #_w1 AND ("DB PUXADOR".REFERENCIAS.FINAL < 0.0) THEN "DB PUXADOR".REFERENCIAS.FINAL := 0.0; END_IF;
   IF "DB PRINCIPAL".AUXILIARES.SEMPRE_1 THEN "Tag_58" := "DB PUXADOR".REFERENCIAS.FINAL - "Tag_56"; END_IF;
   IF "DB PRINCIPAL".AUXILIARES.SEMPRE_1 AND ("Tag_58" > (-1.0)) AND ("Tag_58" < 1.0) THEN
       "DB PUXADOR".REFERENCIAS.FINAL := "Tag_56";
   END_IF;
   IF "DB PRINCIPAL".AUXILIARES.SEMPRE_1 AND NOT "DB PUXADOR".COMANDOS.DESBLOQUEIO_DRIVER AND ("DB PUXADOR".REFERENCIAS.FINAL >= "DB PRINCIPAL".REFERENCIAS.PASSO_DEC) THEN
       "DB PUXADOR".REFERENCIAS.FINAL := "DB PRINCIPAL".REFERENCIAS.PASSO_DEC;
   END_IF;
END_REGION

REGION Network 19: DESBLOQUEIO DO INVERSOR DE FREQUÊNCIA
   // DESBLOQUEIO DO INVERSOR DE FREQUÊNCIA
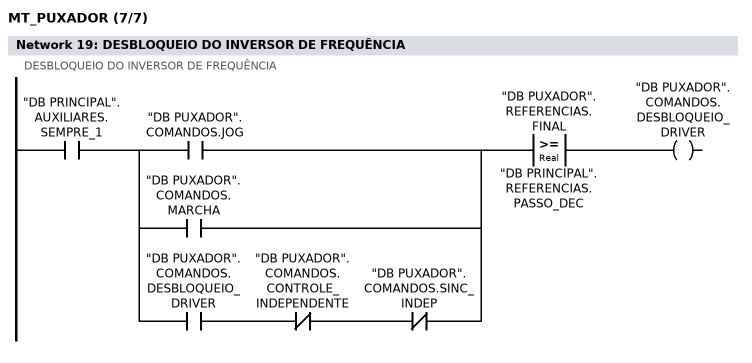
   RUNG wire#powerrail
      Contact( "DB PRINCIPAL".AUXILIARES.SEMPRE_1 )
      wire#w1
      Contact( "DB PUXADOR".COMANDOS.JOG )
      wire#w2
      { S7_Templates := "SrcType := Real" } GE_Contact(in1 := "DB PUXADOR".REFERENCIAS.FINAL, in2 := "DB PRINCIPAL".REFERENCIAS.PASSO_DEC)
      Coil( "DB PUXADOR".COMANDOS.DESBLOQUEIO_DRIVER )
   END_RUNG
   RUNG wire#w1
      Contact( "DB PUXADOR".COMANDOS.MARCHA )
   END_RUNG wire#w2
   RUNG wire#w1
      Contact( "DB PUXADOR".COMANDOS.DESBLOQUEIO_DRIVER )
      I_Contact( "DB PUXADOR".COMANDOS.CONTROLE_INDEPENDENTE )
      I_Contact( "DB PUXADOR".COMANDOS.SINC_INDEP )
   END_RUNG wire#w2
   // the same network as SCL:
   "DB PUXADOR".COMANDOS.DESBLOQUEIO_DRIVER := "DB PRINCIPAL".AUXILIARES.SEMPRE_1 AND ("DB PUXADOR".COMANDOS.JOG OR "DB PUXADOR".COMANDOS.MARCHA OR ("DB PUXADOR".COMANDOS.DESBLOQUEIO_DRIVER AND NOT "DB PUXADOR".COMANDOS.CONTROLE_INDEPENDENTE AND NOT "DB PUXADOR".COMANDOS.SINC_INDEP)) AND ("DB PUXADOR".REFERENCIAS.FINAL >= "DB PRINCIPAL".REFERENCIAS.PASSO_DEC);
END_REGION

REGION Network 20 (STL): STATUS / CONTROLE - INVERSOR DE FREQUÊNCIA
   // DANFOSS FC300 PROFIBUS - TEX24626INV001
   // STATUS DO INVERSOR DE FREQUÊNCIA
         L     "Tag_2":P;
         T     "Tag_1";
         AN    "Tag_59";
         =     "DB PUXADOR".COMANDOS.STATUS_DRIVER;

   // CONTROLE DO INVERSOR DE FREQUÊNCIA
         L     1150;
         T     "Tag_1";
         A     "DB PUXADOR".COMANDOS.DESBLOQUEIO_DRIVER;
         =     "Tag_60";
         A     "T2";
         AN    "DB PUXADOR".COMANDOS.STATUS_DRIVER;
         =     "Tag_61";
         L     "Tag_1";
         T     "Tag_3":P;

   // TRANSFERE A REFERÊNCIA PARA O INVERSOR DE FREQUÊNCIA
         L     "DB PUXADOR".REFERENCIAS.FINAL;
         L     16384.0;
         *R;

         L     "DB PUXADOR".REFERENCIAS.VELOCIDADE_MAXIMA;
         /R;
         RND;
         T     "Tag_62";
         L     "Tag_62";
         T     "Tag_4":P;
END_REGION

REGION Network 21 (STL): INVERSOR RESERVA
         A     "DB PRINCIPAL".AUXILIARES.SEMPRE_1;
         =     %L24.0;
         A     %L24.0;
         A(;
         L     "DB PRINCIPAL".AUXILIARES1.INVERSOR_RESERVA1;
         L     1;
         ==I;
         );
         =     %L24.1;
         A     %L24.1;
         JNB   M001;
         L     "DB PUXADOR".REFERENCIAS.FINAL;
         L     3.456;
         *R;
         T     #aux_r;
         RND;
         T     "P_QW100":P;
   M001: NOP   0;
         A     %L24.1;
         A     "I130";
         S     "DB PRINCIPAL".ALARME.INV_RESERVA1;
         S     "DB PUXADOR".ALARMES.PROTECAO_RESERVA;
         A     %L24.1;
         A     "DB PUXADOR".COMANDOS.DESBLOQUEIO_DRIVER;
         S     "Q134";
         A     %L24.1;
         AN    "DB PUXADOR".COMANDOS.DESBLOQUEIO_DRIVER;
         R     "Q134";
         A     %L24.0;
         A(;
         L     "DB PRINCIPAL".AUXILIARES1.INVERSOR_RESERVA2;
         L     1;
         ==I;
         );
         =     %L24.1;
         A     %L24.1;
         JNB   M002;
         L     "DB PUXADOR".REFERENCIAS.FINAL;
         L     3.456;
         *R;
         T     #aux_r;
         RND;
         T     "P_QW102":P;
   M002: NOP   0;
         A     %L24.1;
         A     "I132";
         S     "DB PRINCIPAL".ALARME.INV_RESERVA2;
         S     "DB PUXADOR".ALARMES.PROTECAO_RESERVA;
         A     %L24.1;
         A     "DB PUXADOR".COMANDOS.DESBLOQUEIO_DRIVER;
         S     "Q135";
         A     %L24.1;
         AN    "DB PUXADOR".COMANDOS.DESBLOQUEIO_DRIVER;
         R     "Q135";
END_REGION
END_FUNCTION

FUNCTION "MT_CHAMUSCADEIRA" : Void   // FC11, LAD
TITLE = MÓDULO DE CONTROLE DA CHAMUSCADEIRA
{ S7_Optimized_Access := 'FALSE' }
AUTHOR : THALLES
FAMILY : TRAÇÃO
NAME : LINHA1
VERSION : 0.1
// DATA BLOCK DE CONTROLE // DB11
// Automation Pack Automação Indl. e Com. Ltda.
// Cliente: Texima S/A Ind. de Máquinas
// Cliente Final: Cia. Fiação e Tecidos Santo Antonio.
// Máquina: LINHA 1 DENIN - O.S.: 24.626
   VAR_TEMP
      AUX_R : Real;
   END_VAR
   VAR_TEMP   // added for the SCL form of the ladder/FBD networks
      _w1 : Bool;
   END_VAR
BEGIN

REGION Network 1: ALARMES
   // RESET DOS ALARMES
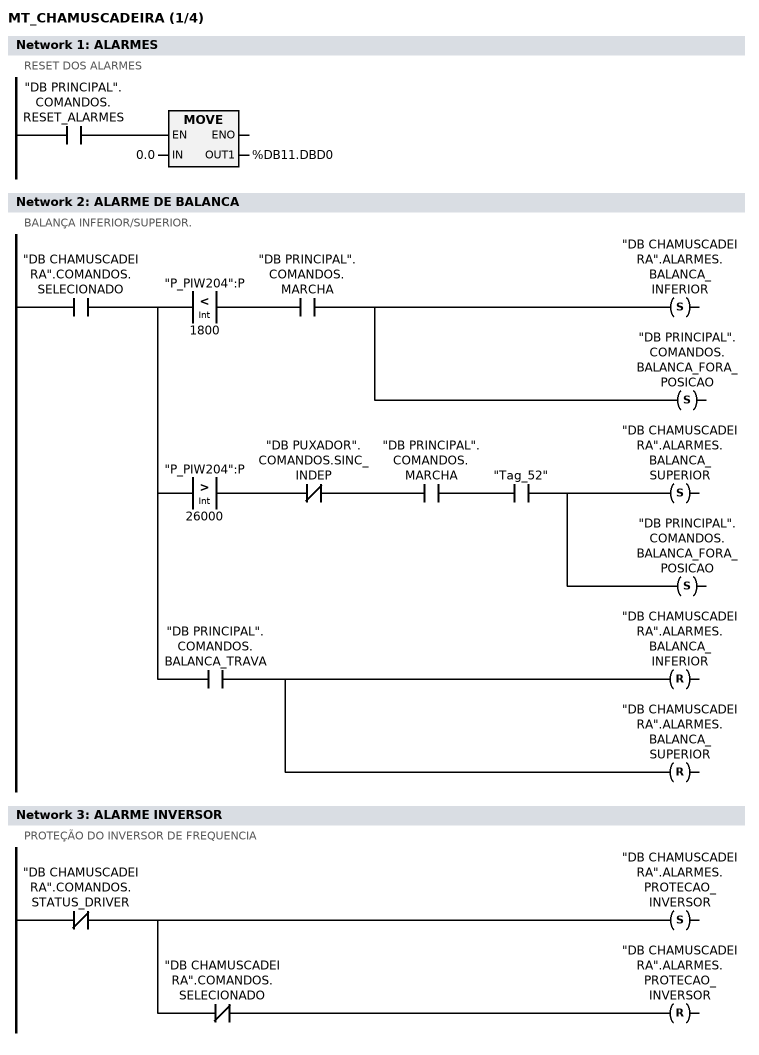
   RUNG wire#powerrail
      Contact( "DB PRINCIPAL".COMANDOS.RESET_ALARMES )
      { S7_GenerateENO := "TRUE" } Move(in := 0.0, out1 => %DB11.DBD0)
   END_RUNG
   // the same network as SCL:
   IF "DB PRINCIPAL".COMANDOS.RESET_ALARMES THEN %DB11.DBD0 := 0.0; END_IF;
END_REGION

REGION Network 2: ALARME DE BALANCA
   // BALANÇA INFERIOR/SUPERIOR.
   RUNG wire#powerrail
      Contact( "DB CHAMUSCADEIRA".COMANDOS.SELECIONADO )
      wire#w1
      { S7_Templates := "SrcType := Int" } LT_Contact(in1 := "P_PIW204":P, in2 := 1800)
      Contact( "DB PRINCIPAL".COMANDOS.MARCHA )
      wire#w2
      S_Coil( "DB CHAMUSCADEIRA".ALARMES.BALANCA_INFERIOR )
   END_RUNG
   RUNG wire#w2
      S_Coil( "DB PRINCIPAL".COMANDOS.BALANCA_FORA_POSICAO )
   END_RUNG
   RUNG wire#w1
      { S7_Templates := "SrcType := Int" } GT_Contact(in1 := "P_PIW204":P, in2 := 26000)
      I_Contact( "DB PUXADOR".COMANDOS.SINC_INDEP )
      Contact( "DB PRINCIPAL".COMANDOS.MARCHA )
      Contact( "Tag_52" )
      wire#w3
      S_Coil( "DB CHAMUSCADEIRA".ALARMES.BALANCA_SUPERIOR )
   END_RUNG
   RUNG wire#w3
      S_Coil( "DB PRINCIPAL".COMANDOS.BALANCA_FORA_POSICAO )
   END_RUNG
   RUNG wire#w1
      Contact( "DB PRINCIPAL".COMANDOS.BALANCA_TRAVA )
      wire#w4
      R_Coil( "DB CHAMUSCADEIRA".ALARMES.BALANCA_INFERIOR )
   END_RUNG
   RUNG wire#w4
      R_Coil( "DB CHAMUSCADEIRA".ALARMES.BALANCA_SUPERIOR )
   END_RUNG
   // the same network as SCL:
   IF "DB CHAMUSCADEIRA".COMANDOS.SELECIONADO AND ("P_PIW204":P < 1800) AND "DB PRINCIPAL".COMANDOS.MARCHA THEN
       "DB CHAMUSCADEIRA".ALARMES.BALANCA_INFERIOR := TRUE;
       "DB PRINCIPAL".COMANDOS.BALANCA_FORA_POSICAO := TRUE;
   END_IF;
   IF "DB CHAMUSCADEIRA".COMANDOS.SELECIONADO AND ("P_PIW204":P > 26000) AND NOT "DB PUXADOR".COMANDOS.SINC_INDEP AND "DB PRINCIPAL".COMANDOS.MARCHA AND "Tag_52" THEN
       "DB CHAMUSCADEIRA".ALARMES.BALANCA_SUPERIOR := TRUE;
       "DB PRINCIPAL".COMANDOS.BALANCA_FORA_POSICAO := TRUE;
   END_IF;
   IF "DB CHAMUSCADEIRA".COMANDOS.SELECIONADO AND "DB PRINCIPAL".COMANDOS.BALANCA_TRAVA THEN
       "DB CHAMUSCADEIRA".ALARMES.BALANCA_INFERIOR := FALSE;
       "DB CHAMUSCADEIRA".ALARMES.BALANCA_SUPERIOR := FALSE;
   END_IF;
END_REGION

REGION Network 3: ALARME INVERSOR
   // PROTEÇÃO DO INVERSOR DE FREQUENCIA
   RUNG wire#powerrail
      I_Contact( "DB CHAMUSCADEIRA".COMANDOS.STATUS_DRIVER )
      wire#w1
      S_Coil( "DB CHAMUSCADEIRA".ALARMES.PROTECAO_INVERSOR )
   END_RUNG
   RUNG wire#w1
      I_Contact( "DB CHAMUSCADEIRA".COMANDOS.SELECIONADO )
      R_Coil( "DB CHAMUSCADEIRA".ALARMES.PROTECAO_INVERSOR )
   END_RUNG
   // the same network as SCL:
   #_w1 := NOT "DB CHAMUSCADEIRA".COMANDOS.STATUS_DRIVER;
   IF #_w1 THEN "DB CHAMUSCADEIRA".ALARMES.PROTECAO_INVERSOR := TRUE; END_IF;
   IF #_w1 AND NOT "DB CHAMUSCADEIRA".COMANDOS.SELECIONADO THEN
       "DB CHAMUSCADEIRA".ALARMES.PROTECAO_INVERSOR := FALSE;
   END_IF;
END_REGION

REGION Network 4: ALARMES
   // ATIVAÇÃO DO BIT DE ALARME DE NIVEL ALTO
   // ATIVAÇÃO DO BIT DE ALARME DE NIVEL BAIXO
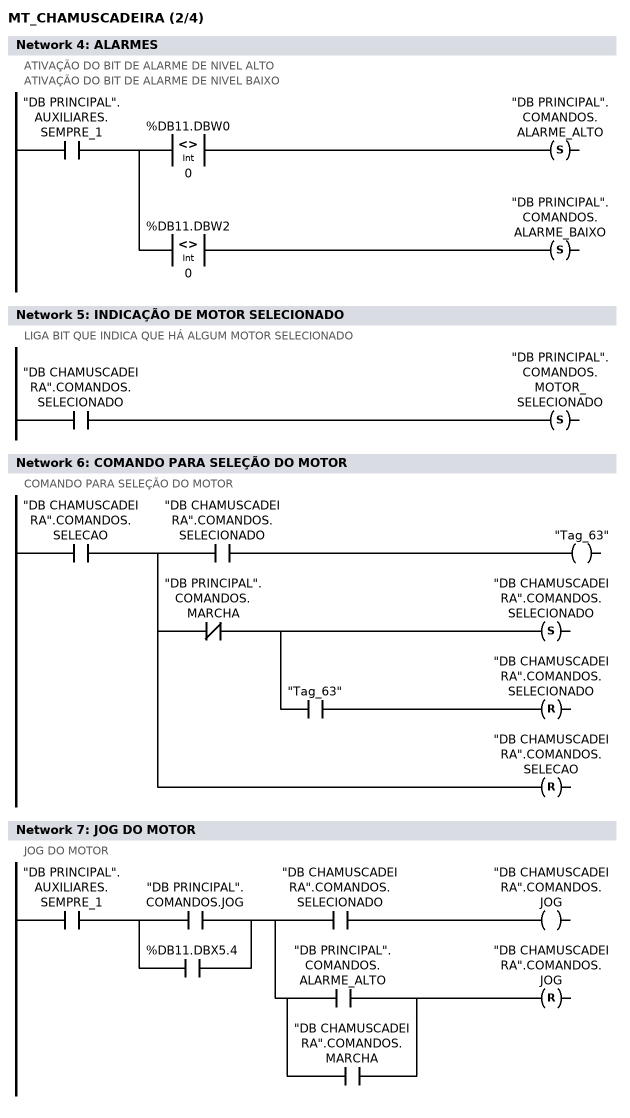
   RUNG wire#powerrail
      Contact( "DB PRINCIPAL".AUXILIARES.SEMPRE_1 )
      wire#w1
      { S7_Templates := "SrcType := Int" } NE_Contact(in1 := %DB11.DBW0, in2 := 0)
      S_Coil( "DB PRINCIPAL".COMANDOS.ALARME_ALTO )
   END_RUNG
   RUNG wire#w1
      { S7_Templates := "SrcType := Int" } NE_Contact(in1 := %DB11.DBW2, in2 := 0)
      S_Coil( "DB PRINCIPAL".COMANDOS.ALARME_BAIXO )
   END_RUNG
   // the same network as SCL:
   IF "DB PRINCIPAL".AUXILIARES.SEMPRE_1 AND (%DB11.DBW0 <> 0) THEN
       "DB PRINCIPAL".COMANDOS.ALARME_ALTO := TRUE;
   END_IF;
   IF "DB PRINCIPAL".AUXILIARES.SEMPRE_1 AND (%DB11.DBW2 <> 0) THEN
       "DB PRINCIPAL".COMANDOS.ALARME_BAIXO := TRUE;
   END_IF;
END_REGION

REGION Network 5: INDICAÇÃO DE MOTOR SELECIONADO
   // LIGA BIT QUE INDICA QUE HÁ ALGUM MOTOR SELECIONADO
   RUNG wire#powerrail
      Contact( "DB CHAMUSCADEIRA".COMANDOS.SELECIONADO )
      S_Coil( "DB PRINCIPAL".COMANDOS.MOTOR_SELECIONADO )
   END_RUNG
   // the same network as SCL:
   IF "DB CHAMUSCADEIRA".COMANDOS.SELECIONADO THEN "DB PRINCIPAL".COMANDOS.MOTOR_SELECIONADO := TRUE; END_IF;
END_REGION

REGION Network 6: COMANDO PARA SELEÇÃO DO MOTOR
   // COMANDO PARA SELEÇÃO DO MOTOR
   RUNG wire#powerrail
      Contact( "DB CHAMUSCADEIRA".COMANDOS.SELECAO )
      wire#w1
      Contact( "DB CHAMUSCADEIRA".COMANDOS.SELECIONADO )
      Coil( "Tag_63" )
   END_RUNG
   RUNG wire#w1
      I_Contact( "DB PRINCIPAL".COMANDOS.MARCHA )
      wire#w2
      S_Coil( "DB CHAMUSCADEIRA".COMANDOS.SELECIONADO )
   END_RUNG
   RUNG wire#w2
      Contact( "Tag_63" )
      R_Coil( "DB CHAMUSCADEIRA".COMANDOS.SELECIONADO )
   END_RUNG
   RUNG wire#w1
      R_Coil( "DB CHAMUSCADEIRA".COMANDOS.SELECAO )
   END_RUNG
   // the same network as SCL:
   "Tag_63" := "DB CHAMUSCADEIRA".COMANDOS.SELECAO AND "DB CHAMUSCADEIRA".COMANDOS.SELECIONADO;
   #_w1 := "DB CHAMUSCADEIRA".COMANDOS.SELECAO AND NOT "DB PRINCIPAL".COMANDOS.MARCHA;
   IF #_w1 THEN "DB CHAMUSCADEIRA".COMANDOS.SELECIONADO := TRUE; END_IF;
   IF #_w1 AND "Tag_63" THEN "DB CHAMUSCADEIRA".COMANDOS.SELECIONADO := FALSE; END_IF;
   IF "DB CHAMUSCADEIRA".COMANDOS.SELECAO THEN "DB CHAMUSCADEIRA".COMANDOS.SELECAO := FALSE; END_IF;
END_REGION

REGION Network 7: JOG DO MOTOR
   // JOG DO MOTOR
   RUNG wire#powerrail
      Contact( "DB PRINCIPAL".AUXILIARES.SEMPRE_1 )
      wire#w1
      Contact( "DB PRINCIPAL".COMANDOS.JOG )
      wire#w2
      Contact( "DB CHAMUSCADEIRA".COMANDOS.SELECIONADO )
      Coil( "DB CHAMUSCADEIRA".COMANDOS.JOG )
   END_RUNG
   RUNG wire#w1
      Contact( %DB11.DBX5.4 )
   END_RUNG wire#w2
   RUNG wire#w2
      Contact( "DB PRINCIPAL".COMANDOS.ALARME_ALTO )
      wire#w3
      R_Coil( "DB CHAMUSCADEIRA".COMANDOS.JOG )
   END_RUNG
   RUNG wire#w2
      Contact( "DB CHAMUSCADEIRA".COMANDOS.MARCHA )
   END_RUNG wire#w3
   // the same network as SCL:
   #_w1 := "DB PRINCIPAL".AUXILIARES.SEMPRE_1 AND ("DB PRINCIPAL".COMANDOS.JOG OR %DB11.DBX5.4);
   "DB CHAMUSCADEIRA".COMANDOS.JOG := #_w1 AND "DB CHAMUSCADEIRA".COMANDOS.SELECIONADO;
   IF #_w1 AND ("DB PRINCIPAL".COMANDOS.ALARME_ALTO OR "DB CHAMUSCADEIRA".COMANDOS.MARCHA) THEN
       "DB CHAMUSCADEIRA".COMANDOS.JOG := FALSE;
   END_IF;
END_REGION

REGION Network 8: COMANDO PARA LIBERAÇÃO DO MOTOR
   // COMANDO PARA LIBERAÇÃO DO MOTOR
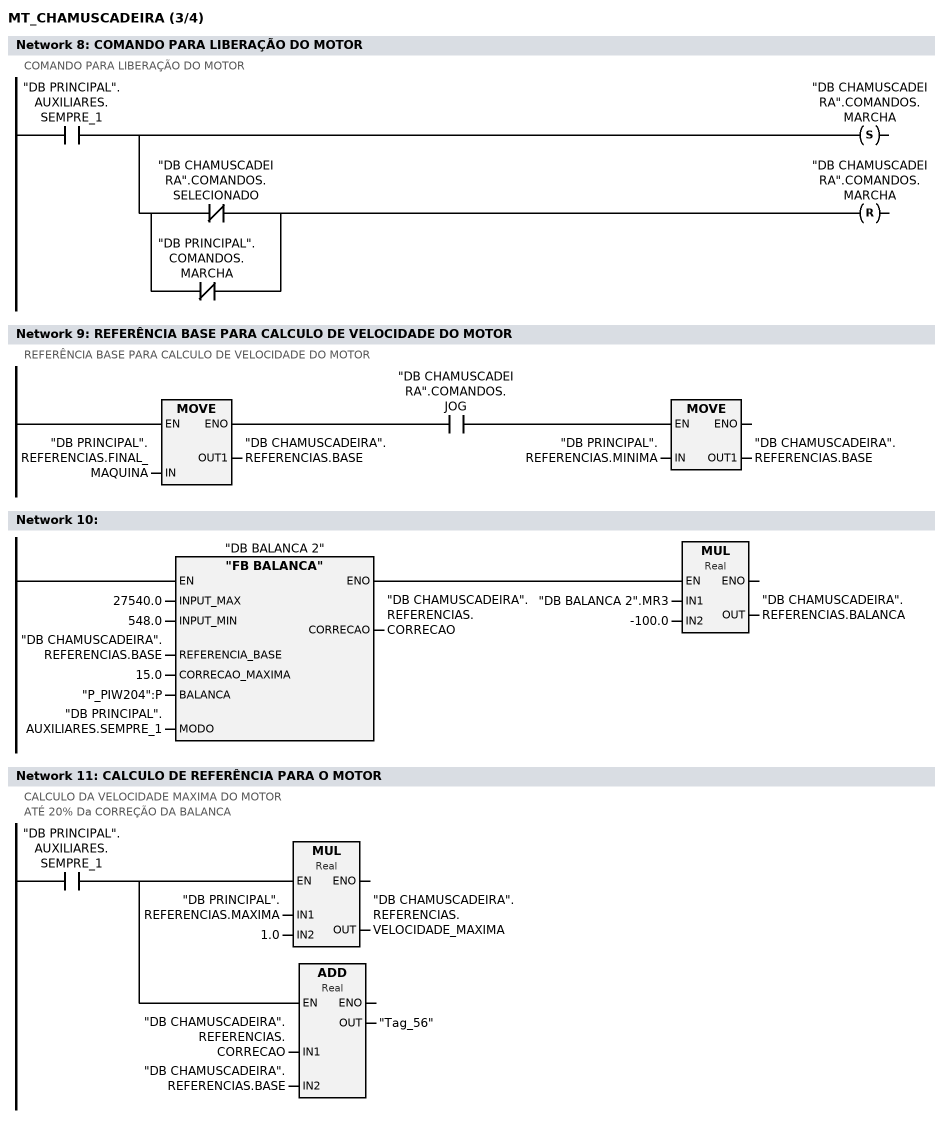
   RUNG wire#powerrail
      Contact( "DB PRINCIPAL".AUXILIARES.SEMPRE_1 )
      wire#w1
      S_Coil( "DB CHAMUSCADEIRA".COMANDOS.MARCHA )
   END_RUNG
   RUNG wire#w1
      I_Contact( "DB CHAMUSCADEIRA".COMANDOS.SELECIONADO )
      wire#w2
      R_Coil( "DB CHAMUSCADEIRA".COMANDOS.MARCHA )
   END_RUNG
   RUNG wire#w1
      I_Contact( "DB PRINCIPAL".COMANDOS.MARCHA )
   END_RUNG wire#w2
   // the same network as SCL:
   IF "DB PRINCIPAL".AUXILIARES.SEMPRE_1 THEN "DB CHAMUSCADEIRA".COMANDOS.MARCHA := TRUE; END_IF;
   IF "DB PRINCIPAL".AUXILIARES.SEMPRE_1 AND (NOT "DB CHAMUSCADEIRA".COMANDOS.SELECIONADO OR NOT "DB PRINCIPAL".COMANDOS.MARCHA) THEN
       "DB CHAMUSCADEIRA".COMANDOS.MARCHA := FALSE;
   END_IF;
END_REGION

REGION Network 9: REFERÊNCIA BASE PARA CALCULO DE VELOCIDADE DO MOTOR
   // REFERÊNCIA BASE PARA CALCULO DE VELOCIDADE DO MOTOR
   RUNG wire#powerrail
      { S7_GenerateENO := "TRUE" } Move(in := "DB PRINCIPAL".REFERENCIAS.FINAL_MAQUINA, out1 => "DB CHAMUSCADEIRA".REFERENCIAS.BASE)
      Contact( "DB CHAMUSCADEIRA".COMANDOS.JOG )
      { S7_GenerateENO := "TRUE" } Move(in := "DB PRINCIPAL".REFERENCIAS.MINIMA, out1 => "DB CHAMUSCADEIRA".REFERENCIAS.BASE)
   END_RUNG
   // the same network as SCL:
   // ENO of a box is taken as its EN; it also drops when the box reports an error
   "DB CHAMUSCADEIRA".REFERENCIAS.BASE := "DB PRINCIPAL".REFERENCIAS.FINAL_MAQUINA;
   IF "DB CHAMUSCADEIRA".COMANDOS.JOG THEN
       "DB CHAMUSCADEIRA".REFERENCIAS.BASE := "DB PRINCIPAL".REFERENCIAS.MINIMA;
   END_IF;
END_REGION

REGION Network 10
   RUNG wire#powerrail
      "DB BALANCA 2"(INPUT_MAX := 27540.0, INPUT_MIN := 548.0, REFERENCIA_BASE := "DB CHAMUSCADEIRA".REFERENCIAS.BASE, CORRECAO_MAXIMA := 15.0, BALANCA := "P_PIW204":P, MODO := "DB PRINCIPAL".AUXILIARES.SEMPRE_1, CORRECAO => "DB CHAMUSCADEIRA".REFERENCIAS.CORRECAO)
      { S7_Templates := "SrcType := Real"; S7_GenerateENO := "TRUE" } Mul(in1 := "DB BALANCA 2".MR3, in2 := -100.0, out => "DB CHAMUSCADEIRA".REFERENCIAS.BALANCA)
   END_RUNG
   // the same network as SCL:
   "DB BALANCA 2"(INPUT_MAX := 27540.0,   // "FB BALANCA"
                  INPUT_MIN := 548.0,
                  REFERENCIA_BASE := "DB CHAMUSCADEIRA".REFERENCIAS.BASE,
                  CORRECAO_MAXIMA := 15.0,
                  BALANCA := "P_PIW204":P,
                  MODO := "DB PRINCIPAL".AUXILIARES.SEMPRE_1,
                  CORRECAO => "DB CHAMUSCADEIRA".REFERENCIAS.CORRECAO,
                  ENO => #_w1);
   IF #_w1 THEN "DB CHAMUSCADEIRA".REFERENCIAS.BALANCA := "DB BALANCA 2".MR3 * (-100.0); END_IF;
END_REGION

REGION Network 11: CALCULO DE REFERÊNCIA PARA O MOTOR
   // CALCULO DA VELOCIDADE MAXIMA DO MOTOR
   // ATÉ 20% Da CORREÇÃO DA BALANCA
   RUNG wire#powerrail
      Contact( "DB PRINCIPAL".AUXILIARES.SEMPRE_1 )
      wire#w1
      { S7_Templates := "SrcType := Real"; S7_GenerateENO := "TRUE" } Mul(in1 := "DB PRINCIPAL".REFERENCIAS.MAXIMA, in2 := 1.0, out => "DB CHAMUSCADEIRA".REFERENCIAS.VELOCIDADE_MAXIMA)
   END_RUNG
   RUNG wire#w1
      { S7_Templates := "SrcType := Real"; S7_GenerateENO := "TRUE" } Add(in1 := "DB CHAMUSCADEIRA".REFERENCIAS.CORRECAO, in2 := "DB CHAMUSCADEIRA".REFERENCIAS.BASE, out => "Tag_56")
   END_RUNG
   // the same network as SCL:
   IF "DB PRINCIPAL".AUXILIARES.SEMPRE_1 THEN
       "DB CHAMUSCADEIRA".REFERENCIAS.VELOCIDADE_MAXIMA := "DB PRINCIPAL".REFERENCIAS.MAXIMA * 1.0;
       "Tag_56" := "DB CHAMUSCADEIRA".REFERENCIAS.CORRECAO + "DB CHAMUSCADEIRA".REFERENCIAS.BASE;
   END_IF;
END_REGION

REGION Network 12
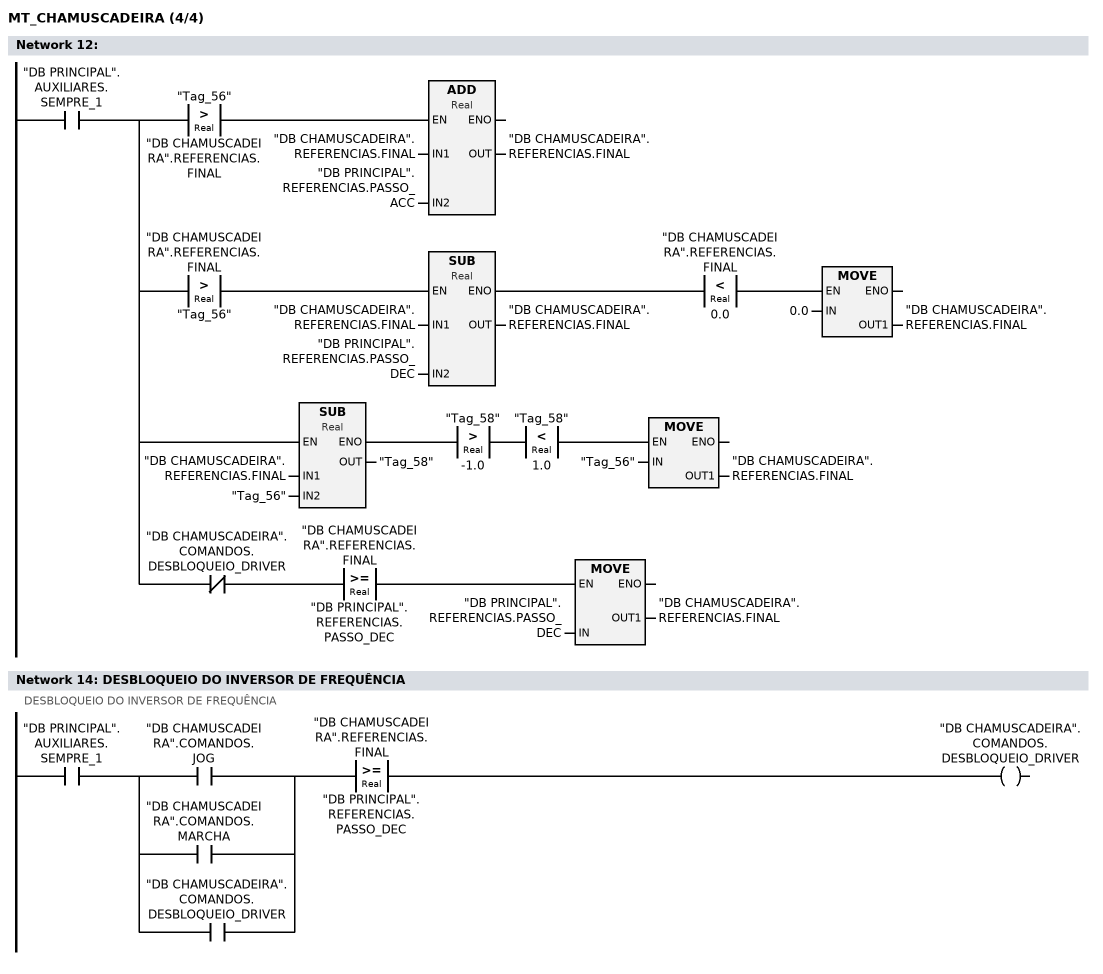
   RUNG wire#powerrail
      Contact( "DB PRINCIPAL".AUXILIARES.SEMPRE_1 )
      wire#w1
      { S7_Templates := "SrcType := Real" } GT_Contact(in1 := "Tag_56", in2 := "DB CHAMUSCADEIRA".REFERENCIAS.FINAL)
      { S7_Templates := "SrcType := Real"; S7_GenerateENO := "TRUE" } Add(in1 := "DB CHAMUSCADEIRA".REFERENCIAS.FINAL, in2 := "DB PRINCIPAL".REFERENCIAS.PASSO_ACC, out => "DB CHAMUSCADEIRA".REFERENCIAS.FINAL)
   END_RUNG
   RUNG wire#w1
      { S7_Templates := "SrcType := Real" } GT_Contact(in1 := "DB CHAMUSCADEIRA".REFERENCIAS.FINAL, in2 := "Tag_56")
      { S7_Templates := "SrcType := Real"; S7_GenerateENO := "TRUE" } Sub(in1 := "DB CHAMUSCADEIRA".REFERENCIAS.FINAL, in2 := "DB PRINCIPAL".REFERENCIAS.PASSO_DEC, out => "DB CHAMUSCADEIRA".REFERENCIAS.FINAL)
      { S7_Templates := "SrcType := Real" } LT_Contact(in1 := "DB CHAMUSCADEIRA".REFERENCIAS.FINAL, in2 := 0.0)
      { S7_GenerateENO := "TRUE" } Move(in := 0.0, out1 => "DB CHAMUSCADEIRA".REFERENCIAS.FINAL)
   END_RUNG
   RUNG wire#w1
      { S7_Templates := "SrcType := Real"; S7_GenerateENO := "TRUE" } Sub(in1 := "DB CHAMUSCADEIRA".REFERENCIAS.FINAL, in2 := "Tag_56", out => "Tag_58")
      { S7_Templates := "SrcType := Real" } GT_Contact(in1 := "Tag_58", in2 := -1.0)
      { S7_Templates := "SrcType := Real" } LT_Contact(in1 := "Tag_58", in2 := 1.0)
      { S7_GenerateENO := "TRUE" } Move(in := "Tag_56", out1 => "DB CHAMUSCADEIRA".REFERENCIAS.FINAL)
   END_RUNG
   RUNG wire#w1
      I_Contact( "DB CHAMUSCADEIRA".COMANDOS.DESBLOQUEIO_DRIVER )
      { S7_Templates := "SrcType := Real" } GE_Contact(in1 := "DB CHAMUSCADEIRA".REFERENCIAS.FINAL, in2 := "DB PRINCIPAL".REFERENCIAS.PASSO_DEC)
      { S7_GenerateENO := "TRUE" } Move(in := "DB PRINCIPAL".REFERENCIAS.PASSO_DEC, out1 => "DB CHAMUSCADEIRA".REFERENCIAS.FINAL)
   END_RUNG
   // the same network as SCL:
   // ENO of a box is taken as its EN; it also drops when the box reports an error
   IF "DB PRINCIPAL".AUXILIARES.SEMPRE_1 AND ("Tag_56" > "DB CHAMUSCADEIRA".REFERENCIAS.FINAL) THEN
       "DB CHAMUSCADEIRA".REFERENCIAS.FINAL := "DB CHAMUSCADEIRA".REFERENCIAS.FINAL + "DB PRINCIPAL".REFERENCIAS.PASSO_ACC;
   END_IF;
   #_w1 := "DB PRINCIPAL".AUXILIARES.SEMPRE_1 AND ("DB CHAMUSCADEIRA".REFERENCIAS.FINAL > "Tag_56");
   IF #_w1 THEN
       "DB CHAMUSCADEIRA".REFERENCIAS.FINAL := "DB CHAMUSCADEIRA".REFERENCIAS.FINAL - "DB PRINCIPAL".REFERENCIAS.PASSO_DEC;
   END_IF;
   IF #_w1 AND ("DB CHAMUSCADEIRA".REFERENCIAS.FINAL < 0.0) THEN
       "DB CHAMUSCADEIRA".REFERENCIAS.FINAL := 0.0;
   END_IF;
   IF "DB PRINCIPAL".AUXILIARES.SEMPRE_1 THEN
       "Tag_58" := "DB CHAMUSCADEIRA".REFERENCIAS.FINAL - "Tag_56";
   END_IF;
   IF "DB PRINCIPAL".AUXILIARES.SEMPRE_1 AND ("Tag_58" > (-1.0)) AND ("Tag_58" < 1.0) THEN
       "DB CHAMUSCADEIRA".REFERENCIAS.FINAL := "Tag_56";
   END_IF;
   IF "DB PRINCIPAL".AUXILIARES.SEMPRE_1 AND NOT "DB CHAMUSCADEIRA".COMANDOS.DESBLOQUEIO_DRIVER AND ("DB CHAMUSCADEIRA".REFERENCIAS.FINAL >= "DB PRINCIPAL".REFERENCIAS.PASSO_DEC) THEN
       "DB CHAMUSCADEIRA".REFERENCIAS.FINAL := "DB PRINCIPAL".REFERENCIAS.PASSO_DEC;
   END_IF;
END_REGION

REGION Network 13 (STL): ACC/DEC DA REFERÊNCIA DO MOTOR
   // ACC/DEC DA REFERÊNCIA DO MOTOR
         A     "DB PRINCIPAL".AUXILIARES.SEMPRE_1;
         =     %L25.0;
         A     %L25.0;
         A(;
         L     "Tag_56";
         L     "DB CHAMUSCADEIRA".REFERENCIAS.FINAL;
         >R;
         );
         JNB   _006;
         L     "DB CHAMUSCADEIRA".REFERENCIAS.FINAL;
         L     "DB PRINCIPAL".REFERENCIAS.PASSO_ACC;
         +R;
         T     "DB CHAMUSCADEIRA".REFERENCIAS.FINAL;
   _006: NOP   0;
         A(;
         A     %L25.0;
         A(;
         L     "DB CHAMUSCADEIRA".REFERENCIAS.FINAL;
         L     "Tag_56";
         >R;
         );
         JNB   _007;
         L     "DB CHAMUSCADEIRA".REFERENCIAS.FINAL;
         L     "DB PRINCIPAL".REFERENCIAS.PASSO_DEC;
         -R;
         T     "DB CHAMUSCADEIRA".REFERENCIAS.FINAL;
         AN    OV;
         SAVE;
         CLR;
   _007: A     BR;
         );
         A(;
         L     "DB CHAMUSCADEIRA".REFERENCIAS.FINAL;
         L     0.0;
         <R;
         );
         JNB   _008;
         L     0.0;
         T     "DB CHAMUSCADEIRA".REFERENCIAS.FINAL;
   _008: NOP   0;
         A(;
         A     %L25.0;
         JNB   _009;
         L     "DB CHAMUSCADEIRA".REFERENCIAS.FINAL;
         L     "Tag_56";
         -R;
         T     "Tag_58";
         AN    OV;
         SAVE;
         CLR;
   _009: A     BR;
         );
         A(;
         L     "Tag_58";
         L     -1.0;
         >R;
         );
         A(;
         L     "Tag_58";
         L     1.0;
         <R;
         );
         JNB   _00a;
         L     "Tag_56";
         T     "DB CHAMUSCADEIRA".REFERENCIAS.FINAL;
   _00a: NOP   0;
         A     %L25.0;
         AN    "DB CHAMUSCADEIRA".COMANDOS.DESBLOQUEIO_DRIVER;
         A(;
         L     "DB CHAMUSCADEIRA".REFERENCIAS.FINAL;
         L     "DB PRINCIPAL".REFERENCIAS.PASSO_DEC;
         >=R;
         );
         JNB   _00b;
         L     "DB PRINCIPAL".REFERENCIAS.PASSO_DEC;
         T     "DB CHAMUSCADEIRA".REFERENCIAS.FINAL;
   _00b: NOP   0;
END_REGION

REGION Network 14: DESBLOQUEIO DO INVERSOR DE FREQUÊNCIA
   // DESBLOQUEIO DO INVERSOR DE FREQUÊNCIA
   RUNG wire#powerrail
      Contact( "DB PRINCIPAL".AUXILIARES.SEMPRE_1 )
      wire#w1
      Contact( "DB CHAMUSCADEIRA".COMANDOS.JOG )
      wire#w2
      { S7_Templates := "SrcType := Real" } GE_Contact(in1 := "DB CHAMUSCADEIRA".REFERENCIAS.FINAL, in2 := "DB PRINCIPAL".REFERENCIAS.PASSO_DEC)
      Coil( "DB CHAMUSCADEIRA".COMANDOS.DESBLOQUEIO_DRIVER )
   END_RUNG
   RUNG wire#w1
      Contact( "DB CHAMUSCADEIRA".COMANDOS.MARCHA )
   END_RUNG wire#w2
   RUNG wire#w1
      Contact( "DB CHAMUSCADEIRA".COMANDOS.DESBLOQUEIO_DRIVER )
   END_RUNG wire#w2
   // the same network as SCL:
   "DB CHAMUSCADEIRA".COMANDOS.DESBLOQUEIO_DRIVER := "DB PRINCIPAL".AUXILIARES.SEMPRE_1 AND ("DB CHAMUSCADEIRA".COMANDOS.JOG OR "DB CHAMUSCADEIRA".COMANDOS.MARCHA OR "DB CHAMUSCADEIRA".COMANDOS.DESBLOQUEIO_DRIVER) AND ("DB CHAMUSCADEIRA".REFERENCIAS.FINAL >= "DB PRINCIPAL".REFERENCIAS.PASSO_DEC);
END_REGION

REGION Network 15 (STL): STATUS / CONTROLE - INVERSOR DE FREQUÊNCIA
   // DANFOSS FC300 PROFIBUS - TEX24626INV001
   // STATUS DO INVERSOR DE FREQUÊNCIA
         L     "Tag_5":P;
         T     "Tag_1";
         AN    "Tag_59";
         =     "DB CHAMUSCADEIRA".COMANDOS.STATUS_DRIVER;

   // CONTROLE DO INVERSOR DE FREQUÊNCIA
         L     1150;
         T     "Tag_1";
         A     "DB CHAMUSCADEIRA".COMANDOS.DESBLOQUEIO_DRIVER;
         =     "Tag_60";
         A     "T2";
         AN    "DB CHAMUSCADEIRA".COMANDOS.STATUS_DRIVER;
         =     "Tag_61";
         L     "Tag_1";
         T     "Tag_6":P;

   // REFERÊNCIA PARA O INVERSOR DE FREQUÊNCIA
         L     "DB CHAMUSCADEIRA".REFERENCIAS.FINAL;
         L     16384.0;
         *R;

         L     "DB CHAMUSCADEIRA".REFERENCIAS.VELOCIDADE_MAXIMA;
         /R;
         RND;
         T     "Tag_62";
         L     "Tag_62";
         T     "Tag_7":P;
END_REGION

REGION Network 16 (STL): INVERSOR RESERVA
         A     "DB PRINCIPAL".AUXILIARES.SEMPRE_1;
         =     %L24.0;
         A     %L24.0;
         A(;
         L     "DB PRINCIPAL".AUXILIARES1.INVERSOR_RESERVA1;
         L     2;
         ==I;
         );
         =     %L24.1;
         A     %L24.1;
         JNB   M00c;
         L     "DB CHAMUSCADEIRA".REFERENCIAS.FINAL;
         L     3.456;
         *R;
         T     #AUX_R;
         RND;
         T     "P_QW100":P;
   M00c: NOP   0;
         A     %L24.1;
         A     "I130";
         S     "DB PRINCIPAL".ALARME.INV_RESERVA1;
         A     %L24.1;
         A     "DB CHAMUSCADEIRA".COMANDOS.DESBLOQUEIO_DRIVER;
         S     "Q134";
         A     %L24.1;
         AN    "DB CHAMUSCADEIRA".COMANDOS.DESBLOQUEIO_DRIVER;
         R     "Q134";
         A     %L24.0;
         A(;
         L     "DB PRINCIPAL".AUXILIARES1.INVERSOR_RESERVA2;
         L     2;
         ==I;
         );
         =     %L24.1;
         A     %L24.1;
         JNB   M00d;
         L     "DB CHAMUSCADEIRA".REFERENCIAS.FINAL;
         L     3.456;
         *R;
         T     #AUX_R;
         RND;
         T     "P_QW102":P;
   M00d: NOP   0;
         A     %L24.1;
         A     "I132";
         S     "DB PRINCIPAL".ALARME.INV_RESERVA2;
         A     %L24.1;
         A     "DB CHAMUSCADEIRA".COMANDOS.DESBLOQUEIO_DRIVER;
         S     "Q135";
         A     %L24.1;
         AN    "DB CHAMUSCADEIRA".COMANDOS.DESBLOQUEIO_DRIVER;
         R     "Q135";
END_REGION
END_FUNCTION

FUNCTION "MT_NEUTRALIZACAO1" : Void   // FC12, LAD
TITLE = MÓDULO DE CONTROLE DA NEUTRALIZACAO 1
{ S7_Optimized_Access := 'FALSE' }
AUTHOR : THALLES
FAMILY : TRAÇÃO
NAME : LINHA1
VERSION : 0.1
// DATA BLOCK DE CONTROLE // DB12
// Automation Pack Automação Indl. e Com. Ltda.
// Cliente: Texima S/A Ind. de Máquinas
// Cliente Final: Cia. Fiação e Tecidos Santo Antonio.
// Máquina: Sanforizadeira SMT-15 - O.S.: 24.626
   VAR_TEMP
      AUX_R : Real;
   END_VAR
   VAR_TEMP   // added for the SCL form of the ladder/FBD networks
      _w1 : Bool;
   END_VAR
BEGIN

REGION Network 1: ALARMES
   // RESET DOS ALARMES
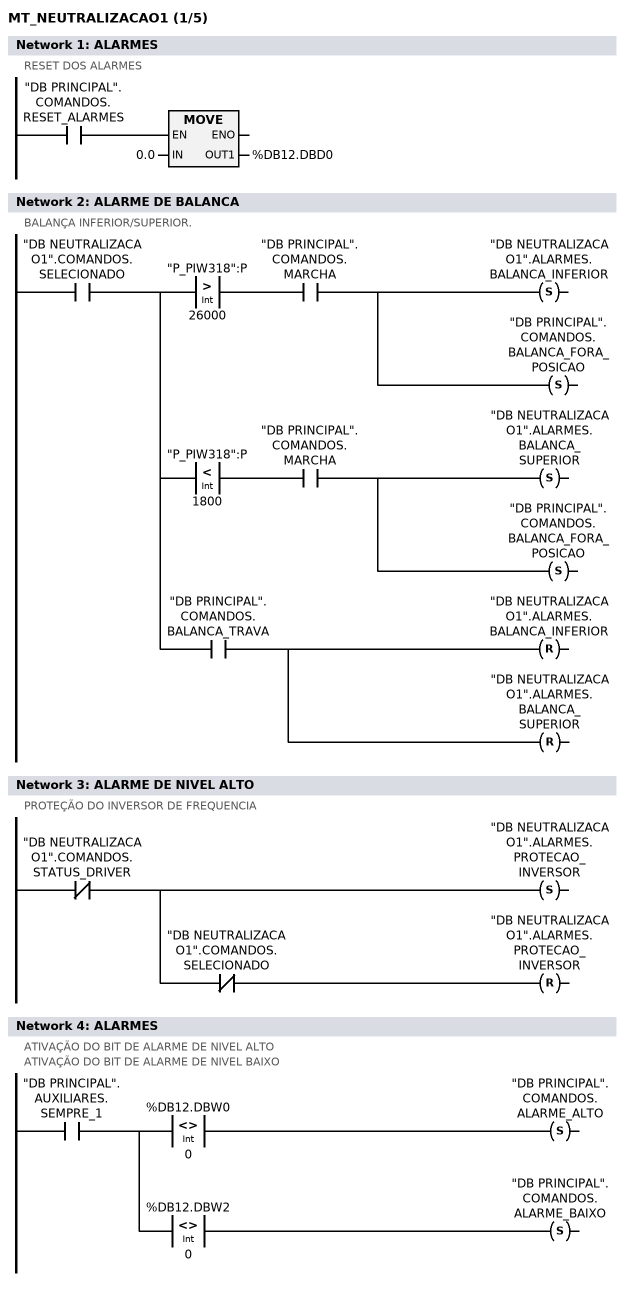
   RUNG wire#powerrail
      Contact( "DB PRINCIPAL".COMANDOS.RESET_ALARMES )
      { S7_GenerateENO := "TRUE" } Move(in := 0.0, out1 => %DB12.DBD0)
   END_RUNG
   // the same network as SCL:
   IF "DB PRINCIPAL".COMANDOS.RESET_ALARMES THEN %DB12.DBD0 := 0.0; END_IF;
END_REGION

REGION Network 2: ALARME DE BALANCA
   // BALANÇA INFERIOR/SUPERIOR.
   RUNG wire#powerrail
      Contact( "DB NEUTRALIZACAO1".COMANDOS.SELECIONADO )
      wire#w1
      { S7_Templates := "SrcType := Int" } GT_Contact(in1 := "P_PIW318":P, in2 := 26000)
      Contact( "DB PRINCIPAL".COMANDOS.MARCHA )
      wire#w2
      S_Coil( "DB NEUTRALIZACAO1".ALARMES.BALANCA_INFERIOR )
   END_RUNG
   RUNG wire#w2
      S_Coil( "DB PRINCIPAL".COMANDOS.BALANCA_FORA_POSICAO )
   END_RUNG
   RUNG wire#w1
      { S7_Templates := "SrcType := Int" } LT_Contact(in1 := "P_PIW318":P, in2 := 1800)
      Contact( "DB PRINCIPAL".COMANDOS.MARCHA )
      wire#w3
      S_Coil( "DB NEUTRALIZACAO1".ALARMES.BALANCA_SUPERIOR )
   END_RUNG
   RUNG wire#w3
      S_Coil( "DB PRINCIPAL".COMANDOS.BALANCA_FORA_POSICAO )
   END_RUNG
   RUNG wire#w1
      Contact( "DB PRINCIPAL".COMANDOS.BALANCA_TRAVA )
      wire#w4
      R_Coil( "DB NEUTRALIZACAO1".ALARMES.BALANCA_INFERIOR )
   END_RUNG
   RUNG wire#w4
      R_Coil( "DB NEUTRALIZACAO1".ALARMES.BALANCA_SUPERIOR )
   END_RUNG
   // the same network as SCL:
   IF "DB NEUTRALIZACAO1".COMANDOS.SELECIONADO AND ("P_PIW318":P > 26000) AND "DB PRINCIPAL".COMANDOS.MARCHA THEN
       "DB NEUTRALIZACAO1".ALARMES.BALANCA_INFERIOR := TRUE;
       "DB PRINCIPAL".COMANDOS.BALANCA_FORA_POSICAO := TRUE;
   END_IF;
   IF "DB NEUTRALIZACAO1".COMANDOS.SELECIONADO AND ("P_PIW318":P < 1800) AND "DB PRINCIPAL".COMANDOS.MARCHA THEN
       "DB NEUTRALIZACAO1".ALARMES.BALANCA_SUPERIOR := TRUE;
       "DB PRINCIPAL".COMANDOS.BALANCA_FORA_POSICAO := TRUE;
   END_IF;
   IF "DB NEUTRALIZACAO1".COMANDOS.SELECIONADO AND "DB PRINCIPAL".COMANDOS.BALANCA_TRAVA THEN
       "DB NEUTRALIZACAO1".ALARMES.BALANCA_INFERIOR := FALSE;
       "DB NEUTRALIZACAO1".ALARMES.BALANCA_SUPERIOR := FALSE;
   END_IF;
END_REGION

REGION Network 3: ALARME DE NIVEL ALTO
   // PROTEÇÃO DO INVERSOR DE FREQUENCIA
   RUNG wire#powerrail
      I_Contact( "DB NEUTRALIZACAO1".COMANDOS.STATUS_DRIVER )
      wire#w1
      S_Coil( "DB NEUTRALIZACAO1".ALARMES.PROTECAO_INVERSOR )
   END_RUNG
   RUNG wire#w1
      I_Contact( "DB NEUTRALIZACAO1".COMANDOS.SELECIONADO )
      R_Coil( "DB NEUTRALIZACAO1".ALARMES.PROTECAO_INVERSOR )
   END_RUNG
   // the same network as SCL:
   #_w1 := NOT "DB NEUTRALIZACAO1".COMANDOS.STATUS_DRIVER;
   IF #_w1 THEN "DB NEUTRALIZACAO1".ALARMES.PROTECAO_INVERSOR := TRUE; END_IF;
   IF #_w1 AND NOT "DB NEUTRALIZACAO1".COMANDOS.SELECIONADO THEN
       "DB NEUTRALIZACAO1".ALARMES.PROTECAO_INVERSOR := FALSE;
   END_IF;
END_REGION

REGION Network 4: ALARMES
   // ATIVAÇÃO DO BIT DE ALARME DE NIVEL ALTO
   // ATIVAÇÃO DO BIT DE ALARME DE NIVEL BAIXO
   RUNG wire#powerrail
      Contact( "DB PRINCIPAL".AUXILIARES.SEMPRE_1 )
      wire#w1
      { S7_Templates := "SrcType := Int" } NE_Contact(in1 := %DB12.DBW0, in2 := 0)
      S_Coil( "DB PRINCIPAL".COMANDOS.ALARME_ALTO )
   END_RUNG
   RUNG wire#w1
      { S7_Templates := "SrcType := Int" } NE_Contact(in1 := %DB12.DBW2, in2 := 0)
      S_Coil( "DB PRINCIPAL".COMANDOS.ALARME_BAIXO )
   END_RUNG
   // the same network as SCL:
   IF "DB PRINCIPAL".AUXILIARES.SEMPRE_1 AND (%DB12.DBW0 <> 0) THEN
       "DB PRINCIPAL".COMANDOS.ALARME_ALTO := TRUE;
   END_IF;
   IF "DB PRINCIPAL".AUXILIARES.SEMPRE_1 AND (%DB12.DBW2 <> 0) THEN
       "DB PRINCIPAL".COMANDOS.ALARME_BAIXO := TRUE;
   END_IF;
END_REGION

REGION Network 5: INDICAÇÃO DE MOTOR SELECIONADO
   // LIGA BIT QUE INDICA QUE HÁ ALGUM MOTOR SELECIONADO
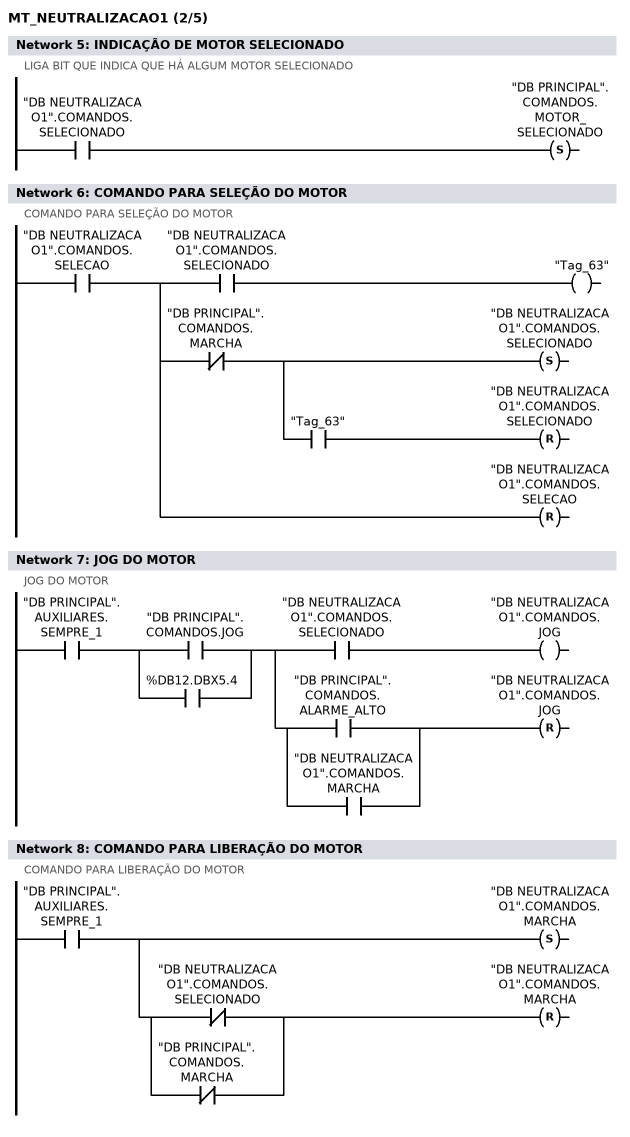
   RUNG wire#powerrail
      Contact( "DB NEUTRALIZACAO1".COMANDOS.SELECIONADO )
      S_Coil( "DB PRINCIPAL".COMANDOS.MOTOR_SELECIONADO )
   END_RUNG
   // the same network as SCL:
   IF "DB NEUTRALIZACAO1".COMANDOS.SELECIONADO THEN
       "DB PRINCIPAL".COMANDOS.MOTOR_SELECIONADO := TRUE;
   END_IF;
END_REGION

REGION Network 6: COMANDO PARA SELEÇÃO DO MOTOR
   // COMANDO PARA SELEÇÃO DO MOTOR
   RUNG wire#powerrail
      Contact( "DB NEUTRALIZACAO1".COMANDOS.SELECAO )
      wire#w1
      Contact( "DB NEUTRALIZACAO1".COMANDOS.SELECIONADO )
      Coil( "Tag_63" )
   END_RUNG
   RUNG wire#w1
      I_Contact( "DB PRINCIPAL".COMANDOS.MARCHA )
      wire#w2
      S_Coil( "DB NEUTRALIZACAO1".COMANDOS.SELECIONADO )
   END_RUNG
   RUNG wire#w2
      Contact( "Tag_63" )
      R_Coil( "DB NEUTRALIZACAO1".COMANDOS.SELECIONADO )
   END_RUNG
   RUNG wire#w1
      R_Coil( "DB NEUTRALIZACAO1".COMANDOS.SELECAO )
   END_RUNG
   // the same network as SCL:
   "Tag_63" := "DB NEUTRALIZACAO1".COMANDOS.SELECAO AND "DB NEUTRALIZACAO1".COMANDOS.SELECIONADO;
   #_w1 := "DB NEUTRALIZACAO1".COMANDOS.SELECAO AND NOT "DB PRINCIPAL".COMANDOS.MARCHA;
   IF #_w1 THEN "DB NEUTRALIZACAO1".COMANDOS.SELECIONADO := TRUE; END_IF;
   IF #_w1 AND "Tag_63" THEN "DB NEUTRALIZACAO1".COMANDOS.SELECIONADO := FALSE; END_IF;
   IF "DB NEUTRALIZACAO1".COMANDOS.SELECAO THEN "DB NEUTRALIZACAO1".COMANDOS.SELECAO := FALSE; END_IF;
END_REGION

REGION Network 7: JOG DO MOTOR
   // JOG DO MOTOR
   RUNG wire#powerrail
      Contact( "DB PRINCIPAL".AUXILIARES.SEMPRE_1 )
      wire#w1
      Contact( "DB PRINCIPAL".COMANDOS.JOG )
      wire#w2
      Contact( "DB NEUTRALIZACAO1".COMANDOS.SELECIONADO )
      Coil( "DB NEUTRALIZACAO1".COMANDOS.JOG )
   END_RUNG
   RUNG wire#w1
      Contact( %DB12.DBX5.4 )
   END_RUNG wire#w2
   RUNG wire#w2
      Contact( "DB PRINCIPAL".COMANDOS.ALARME_ALTO )
      wire#w3
      R_Coil( "DB NEUTRALIZACAO1".COMANDOS.JOG )
   END_RUNG
   RUNG wire#w2
      Contact( "DB NEUTRALIZACAO1".COMANDOS.MARCHA )
   END_RUNG wire#w3
   // the same network as SCL:
   #_w1 := "DB PRINCIPAL".AUXILIARES.SEMPRE_1 AND ("DB PRINCIPAL".COMANDOS.JOG OR %DB12.DBX5.4);
   "DB NEUTRALIZACAO1".COMANDOS.JOG := #_w1 AND "DB NEUTRALIZACAO1".COMANDOS.SELECIONADO;
   IF #_w1 AND ("DB PRINCIPAL".COMANDOS.ALARME_ALTO OR "DB NEUTRALIZACAO1".COMANDOS.MARCHA) THEN
       "DB NEUTRALIZACAO1".COMANDOS.JOG := FALSE;
   END_IF;
END_REGION

REGION Network 8: COMANDO PARA LIBERAÇÃO DO MOTOR
   // COMANDO PARA LIBERAÇÃO DO MOTOR
   RUNG wire#powerrail
      Contact( "DB PRINCIPAL".AUXILIARES.SEMPRE_1 )
      wire#w1
      S_Coil( "DB NEUTRALIZACAO1".COMANDOS.MARCHA )
   END_RUNG
   RUNG wire#w1
      I_Contact( "DB NEUTRALIZACAO1".COMANDOS.SELECIONADO )
      wire#w2
      R_Coil( "DB NEUTRALIZACAO1".COMANDOS.MARCHA )
   END_RUNG
   RUNG wire#w1
      I_Contact( "DB PRINCIPAL".COMANDOS.MARCHA )
   END_RUNG wire#w2
   // the same network as SCL:
   IF "DB PRINCIPAL".AUXILIARES.SEMPRE_1 THEN "DB NEUTRALIZACAO1".COMANDOS.MARCHA := TRUE; END_IF;
   IF "DB PRINCIPAL".AUXILIARES.SEMPRE_1 AND (NOT "DB NEUTRALIZACAO1".COMANDOS.SELECIONADO OR NOT "DB PRINCIPAL".COMANDOS.MARCHA) THEN
       "DB NEUTRALIZACAO1".COMANDOS.MARCHA := FALSE;
   END_IF;
END_REGION

REGION Network 9
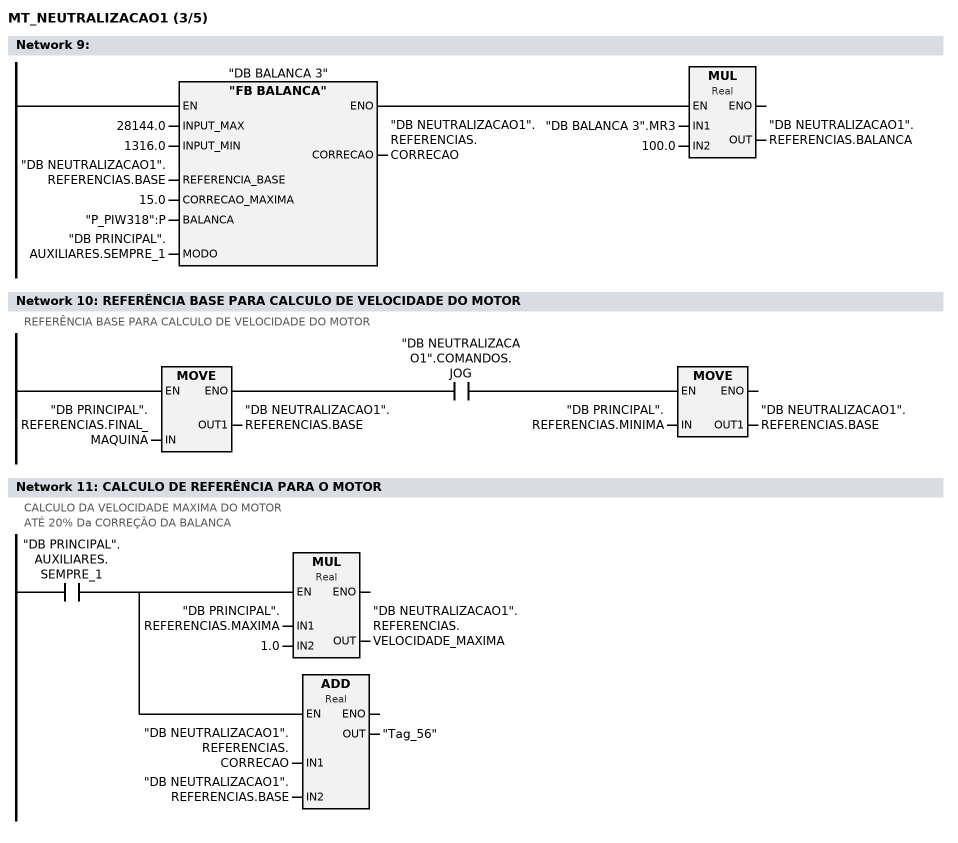
   RUNG wire#powerrail
      "DB BALANCA 3"(INPUT_MAX := 28144.0, INPUT_MIN := 1316.0, REFERENCIA_BASE := "DB NEUTRALIZACAO1".REFERENCIAS.BASE, CORRECAO_MAXIMA := 15.0, BALANCA := "P_PIW318":P, MODO := "DB PRINCIPAL".AUXILIARES.SEMPRE_1, CORRECAO => "DB NEUTRALIZACAO1".REFERENCIAS.CORRECAO)
      { S7_Templates := "SrcType := Real"; S7_GenerateENO := "TRUE" } Mul(in1 := "DB BALANCA 3".MR3, in2 := 100.0, out => "DB NEUTRALIZACAO1".REFERENCIAS.BALANCA)
   END_RUNG
   // the same network as SCL:
   "DB BALANCA 3"(INPUT_MAX := 28144.0,   // "FB BALANCA"
                  INPUT_MIN := 1316.0,
                  REFERENCIA_BASE := "DB NEUTRALIZACAO1".REFERENCIAS.BASE,
                  CORRECAO_MAXIMA := 15.0,
                  BALANCA := "P_PIW318":P,
                  MODO := "DB PRINCIPAL".AUXILIARES.SEMPRE_1,
                  CORRECAO => "DB NEUTRALIZACAO1".REFERENCIAS.CORRECAO,
                  ENO => #_w1);
   IF #_w1 THEN "DB NEUTRALIZACAO1".REFERENCIAS.BALANCA := "DB BALANCA 3".MR3 * 100.0; END_IF;
END_REGION

REGION Network 10: REFERÊNCIA BASE PARA CALCULO DE VELOCIDADE DO MOTOR
   // REFERÊNCIA BASE PARA CALCULO DE VELOCIDADE DO MOTOR
   RUNG wire#powerrail
      { S7_GenerateENO := "TRUE" } Move(in := "DB PRINCIPAL".REFERENCIAS.FINAL_MAQUINA, out1 => "DB NEUTRALIZACAO1".REFERENCIAS.BASE)
      Contact( "DB NEUTRALIZACAO1".COMANDOS.JOG )
      { S7_GenerateENO := "TRUE" } Move(in := "DB PRINCIPAL".REFERENCIAS.MINIMA, out1 => "DB NEUTRALIZACAO1".REFERENCIAS.BASE)
   END_RUNG
   // the same network as SCL:
   // ENO of a box is taken as its EN; it also drops when the box reports an error
   "DB NEUTRALIZACAO1".REFERENCIAS.BASE := "DB PRINCIPAL".REFERENCIAS.FINAL_MAQUINA;
   IF "DB NEUTRALIZACAO1".COMANDOS.JOG THEN
       "DB NEUTRALIZACAO1".REFERENCIAS.BASE := "DB PRINCIPAL".REFERENCIAS.MINIMA;
   END_IF;
END_REGION

REGION Network 11: CALCULO DE REFERÊNCIA PARA O MOTOR
   // CALCULO DA VELOCIDADE MAXIMA DO MOTOR
   // ATÉ 20% Da CORREÇÃO DA BALANCA
   RUNG wire#powerrail
      Contact( "DB PRINCIPAL".AUXILIARES.SEMPRE_1 )
      wire#w1
      { S7_Templates := "SrcType := Real"; S7_GenerateENO := "TRUE" } Mul(in1 := "DB PRINCIPAL".REFERENCIAS.MAXIMA, in2 := 1.0, out => "DB NEUTRALIZACAO1".REFERENCIAS.VELOCIDADE_MAXIMA)
   END_RUNG
   RUNG wire#w1
      { S7_Templates := "SrcType := Real"; S7_GenerateENO := "TRUE" } Add(in1 := "DB NEUTRALIZACAO1".REFERENCIAS.CORRECAO, in2 := "DB NEUTRALIZACAO1".REFERENCIAS.BASE, out => "Tag_56")
   END_RUNG
   // the same network as SCL:
   IF "DB PRINCIPAL".AUXILIARES.SEMPRE_1 THEN
       "DB NEUTRALIZACAO1".REFERENCIAS.VELOCIDADE_MAXIMA := "DB PRINCIPAL".REFERENCIAS.MAXIMA * 1.0;
       "Tag_56" := "DB NEUTRALIZACAO1".REFERENCIAS.CORRECAO + "DB NEUTRALIZACAO1".REFERENCIAS.BASE;
   END_IF;
END_REGION

REGION Network 12: ACC/DEC DA REFERÊNCIA DO MOTOR
   // ACC/DEC DA REFERÊNCIA DO MOTOR
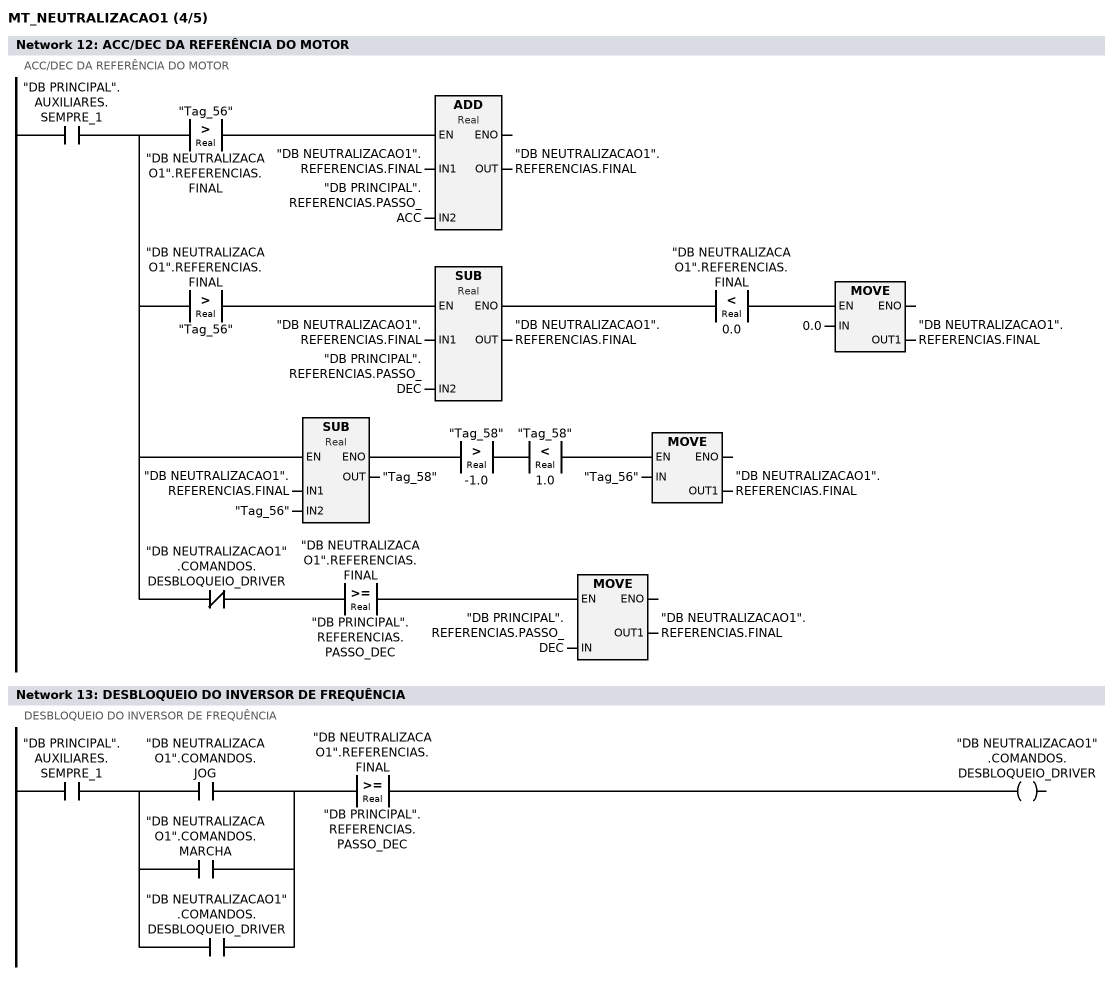
   RUNG wire#powerrail
      Contact( "DB PRINCIPAL".AUXILIARES.SEMPRE_1 )
      wire#w1
      { S7_Templates := "SrcType := Real" } GT_Contact(in1 := "Tag_56", in2 := "DB NEUTRALIZACAO1".REFERENCIAS.FINAL)
      { S7_Templates := "SrcType := Real"; S7_GenerateENO := "TRUE" } Add(in1 := "DB NEUTRALIZACAO1".REFERENCIAS.FINAL, in2 := "DB PRINCIPAL".REFERENCIAS.PASSO_ACC, out => "DB NEUTRALIZACAO1".REFERENCIAS.FINAL)
   END_RUNG
   RUNG wire#w1
      { S7_Templates := "SrcType := Real" } GT_Contact(in1 := "DB NEUTRALIZACAO1".REFERENCIAS.FINAL, in2 := "Tag_56")
      { S7_Templates := "SrcType := Real"; S7_GenerateENO := "TRUE" } Sub(in1 := "DB NEUTRALIZACAO1".REFERENCIAS.FINAL, in2 := "DB PRINCIPAL".REFERENCIAS.PASSO_DEC, out => "DB NEUTRALIZACAO1".REFERENCIAS.FINAL)
      { S7_Templates := "SrcType := Real" } LT_Contact(in1 := "DB NEUTRALIZACAO1".REFERENCIAS.FINAL, in2 := 0.0)
      { S7_GenerateENO := "TRUE" } Move(in := 0.0, out1 => "DB NEUTRALIZACAO1".REFERENCIAS.FINAL)
   END_RUNG
   RUNG wire#w1
      { S7_Templates := "SrcType := Real"; S7_GenerateENO := "TRUE" } Sub(in1 := "DB NEUTRALIZACAO1".REFERENCIAS.FINAL, in2 := "Tag_56", out => "Tag_58")
      { S7_Templates := "SrcType := Real" } GT_Contact(in1 := "Tag_58", in2 := -1.0)
      { S7_Templates := "SrcType := Real" } LT_Contact(in1 := "Tag_58", in2 := 1.0)
      { S7_GenerateENO := "TRUE" } Move(in := "Tag_56", out1 => "DB NEUTRALIZACAO1".REFERENCIAS.FINAL)
   END_RUNG
   RUNG wire#w1
      I_Contact( "DB NEUTRALIZACAO1".COMANDOS.DESBLOQUEIO_DRIVER )
      { S7_Templates := "SrcType := Real" } GE_Contact(in1 := "DB NEUTRALIZACAO1".REFERENCIAS.FINAL, in2 := "DB PRINCIPAL".REFERENCIAS.PASSO_DEC)
      { S7_GenerateENO := "TRUE" } Move(in := "DB PRINCIPAL".REFERENCIAS.PASSO_DEC, out1 => "DB NEUTRALIZACAO1".REFERENCIAS.FINAL)
   END_RUNG
   // the same network as SCL:
   // ENO of a box is taken as its EN; it also drops when the box reports an error
   IF "DB PRINCIPAL".AUXILIARES.SEMPRE_1 AND ("Tag_56" > "DB NEUTRALIZACAO1".REFERENCIAS.FINAL) THEN
       "DB NEUTRALIZACAO1".REFERENCIAS.FINAL := "DB NEUTRALIZACAO1".REFERENCIAS.FINAL + "DB PRINCIPAL".REFERENCIAS.PASSO_ACC;
   END_IF;
   #_w1 := "DB PRINCIPAL".AUXILIARES.SEMPRE_1 AND ("DB NEUTRALIZACAO1".REFERENCIAS.FINAL > "Tag_56");
   IF #_w1 THEN
       "DB NEUTRALIZACAO1".REFERENCIAS.FINAL := "DB NEUTRALIZACAO1".REFERENCIAS.FINAL - "DB PRINCIPAL".REFERENCIAS.PASSO_DEC;
   END_IF;
   IF #_w1 AND ("DB NEUTRALIZACAO1".REFERENCIAS.FINAL < 0.0) THEN
       "DB NEUTRALIZACAO1".REFERENCIAS.FINAL := 0.0;
   END_IF;
   IF "DB PRINCIPAL".AUXILIARES.SEMPRE_1 THEN
       "Tag_58" := "DB NEUTRALIZACAO1".REFERENCIAS.FINAL - "Tag_56";
   END_IF;
   IF "DB PRINCIPAL".AUXILIARES.SEMPRE_1 AND ("Tag_58" > (-1.0)) AND ("Tag_58" < 1.0) THEN
       "DB NEUTRALIZACAO1".REFERENCIAS.FINAL := "Tag_56";
   END_IF;
   IF "DB PRINCIPAL".AUXILIARES.SEMPRE_1 AND NOT "DB NEUTRALIZACAO1".COMANDOS.DESBLOQUEIO_DRIVER AND ("DB NEUTRALIZACAO1".REFERENCIAS.FINAL >= "DB PRINCIPAL".REFERENCIAS.PASSO_DEC) THEN
       "DB NEUTRALIZACAO1".REFERENCIAS.FINAL := "DB PRINCIPAL".REFERENCIAS.PASSO_DEC;
   END_IF;
END_REGION

REGION Network 13: DESBLOQUEIO DO INVERSOR DE FREQUÊNCIA
   // DESBLOQUEIO DO INVERSOR DE FREQUÊNCIA
   RUNG wire#powerrail
      Contact( "DB PRINCIPAL".AUXILIARES.SEMPRE_1 )
      wire#w1
      Contact( "DB NEUTRALIZACAO1".COMANDOS.JOG )
      wire#w2
      { S7_Templates := "SrcType := Real" } GE_Contact(in1 := "DB NEUTRALIZACAO1".REFERENCIAS.FINAL, in2 := "DB PRINCIPAL".REFERENCIAS.PASSO_DEC)
      Coil( "DB NEUTRALIZACAO1".COMANDOS.DESBLOQUEIO_DRIVER )
   END_RUNG
   RUNG wire#w1
      Contact( "DB NEUTRALIZACAO1".COMANDOS.MARCHA )
   END_RUNG wire#w2
   RUNG wire#w1
      Contact( "DB NEUTRALIZACAO1".COMANDOS.DESBLOQUEIO_DRIVER )
   END_RUNG wire#w2
   // the same network as SCL:
   "DB NEUTRALIZACAO1".COMANDOS.DESBLOQUEIO_DRIVER := "DB PRINCIPAL".AUXILIARES.SEMPRE_1 AND ("DB NEUTRALIZACAO1".COMANDOS.JOG OR "DB NEUTRALIZACAO1".COMANDOS.MARCHA OR "DB NEUTRALIZACAO1".COMANDOS.DESBLOQUEIO_DRIVER) AND ("DB NEUTRALIZACAO1".REFERENCIAS.FINAL >= "DB PRINCIPAL".REFERENCIAS.PASSO_DEC);
END_REGION

REGION Network 14 (STL): STATUS / CONTROLE - INVERSOR DE FREQUÊNCIA
   // DANFOSS FC300 PROFIBUS - TEX24626INV001
   // STATUS DO INVERSOR DE FREQUÊNCIA
         L     "Tag_8":P;
         T     "Tag_1";
         AN    "Tag_59";
         =     "DB NEUTRALIZACAO1".COMANDOS.STATUS_DRIVER;

   // CONTROLE DO INVERSOR DE FREQUÊNCIA
         L     1150;
         T     "Tag_1";
         A     "DB NEUTRALIZACAO1".COMANDOS.DESBLOQUEIO_DRIVER;
         =     "Tag_60";
         A     "T2";
         AN    "DB NEUTRALIZACAO1".COMANDOS.STATUS_DRIVER;
         =     "Tag_61";
         L     "Tag_1";
         T     "Tag_9":P;

   // REFERÊNCIA PARA O INVERSOR DE FREQUÊNCIA
         L     "DB NEUTRALIZACAO1".REFERENCIAS.FINAL;
         L     16384.0;
         *R;

         L     "DB NEUTRALIZACAO1".REFERENCIAS.VELOCIDADE_MAXIMA;
         /R;
         RND;
         T     "Tag_62";
         L     "Tag_62";
         T     "Tag_10":P;
END_REGION

REGION Network 15 (STL): INVERSOR RESERVA
         A     "DB PRINCIPAL".AUXILIARES.SEMPRE_1;
         =     %L24.0;
         A     %L24.0;
         A(;
         L     "DB PRINCIPAL".AUXILIARES1.INVERSOR_RESERVA1;
         L     3;
         ==I;
         );
         =     %L24.1;
         A     %L24.1;
         JNB   M001;
         L     "DB NEUTRALIZACAO1".REFERENCIAS.FINAL;
         L     3.456;
         *R;
         T     #AUX_R;
         RND;
         T     "P_QW100":P;
   M001: NOP   0;
         A     %L24.1;
         A     "I130";
         S     "DB PRINCIPAL".ALARME.INV_RESERVA1;
         A     %L24.1;
         A     "DB NEUTRALIZACAO1".COMANDOS.DESBLOQUEIO_DRIVER;
         S     "Q134";
         A     %L24.1;
         AN    "DB NEUTRALIZACAO1".COMANDOS.DESBLOQUEIO_DRIVER;
         R     "Q134";
         A     %L24.0;
         A(;
         L     "DB PRINCIPAL".AUXILIARES1.INVERSOR_RESERVA2;
         L     3;
         ==I;
         );
         =     %L24.1;
         A     %L24.1;
         JNB   M002;
         L     "DB NEUTRALIZACAO1".REFERENCIAS.FINAL;
         L     3.456;
         *R;
         T     #AUX_R;
         RND;
         T     "P_QW102":P;
   M002: NOP   0;
         A     %L24.1;
         A     "I132";
         S     "DB PRINCIPAL".ALARME.INV_RESERVA2;
         A     %L24.1;
         A     "DB NEUTRALIZACAO1".COMANDOS.DESBLOQUEIO_DRIVER;
         S     "Q135";
         A     %L24.1;
         AN    "DB NEUTRALIZACAO1".COMANDOS.DESBLOQUEIO_DRIVER;
         R     "Q135";
END_REGION

REGION Network 16
